_stTmp.rMasterPos           := _mcMotionFunctionPoint.MasterPos;
_stTmp.rSlavePos            := _mcMotionFunctionPoint.SlavePos;
_stTmp.rSlaveAcc            := _mcMotionFunctionPoint.SlaveAcc;
_stTmp.rSlaveJerk           := _mcMotionFunctionPoint.SlaveJerk;
_stTmp.rSlaveVelo           := _mcMotionFunctionPoint.SlaveVelo;

ReadMotionFunctionPointData := _stTmp;
END_GET
END_PROPERTY

METHOD ReadMotionFunctionValues : E_PROGRESS
VAR_INPUT
  Execute           : BOOL;
END_VAR
VAR_INST
  _eState           : E_PROGRESS;
  _rValue           : LREAL;
  _udiErr           : UDINT;
  _stMsg            : ST_Message;
END_VAR

IF NOT Execute THEN _eState   := E_PROGRESS.INIT; END_IF


CASE _eState
OF
  E_PROGRESS.INIT:
    IF Execute 
    THEN
      memset(ADR(_mcMotionFunction),0,SIZEOF(_mcMotionFunction));
      memset(ADR(_stMsg),0,SIZEOF(_stMsg));
      _udiErr                       := 0;
      _rValue                       := 0;
      _eState                       := E_PROGRESS.BUSY;

      _mcCamRef.pArray              := ADR(_mcMotionFunction);
      _mcCamRef.ArraySize           := SIZEOF(_mcMotionFunction);

      _mcCamRef.TableType           := Tc2_MC2_Camming.MC_TABLETYPE_MOTIONFUNCTION;
      _mcCamRef.NoOfColumns         := 1;

      _fbReadMotionFunctionValues(
              Execute               := FALSE, 
              CamTableID            := _stCamData.nCamTableId, 
              ValueSelectMask       := _stCamData.stReadValuesParameter.nValueSelectMask, 
              StartPosMaster        := _stCamData.stReadValuesParameter.rValueMasterStart, 
              EndPosMaster          := _stCamData.stReadValuesParameter.rValueMasterEnd, 
              Increment             := _stCamData.stReadValuesParameter.rIncrement, 
              CamTable              := _mcCamRef);
    END_IF
END_CASE
CASE _eState
OF
  E_PROGRESS.BUSY:
    _fbReadMotionFunctionValues(
              Execute               := TRUE, 
              CamTableID            := _stCamData.nCamTableId, 
              ValueSelectMask       := _stCamData.stReadValuesParameter.nValueSelectMask, 
              StartPosMaster        := _stCamData.stReadValuesParameter.rValueMasterStart, 
              EndPosMaster          := _stCamData.stReadValuesParameter.rValueMasterEnd, 
              Increment             := _stCamData.stReadValuesParameter.rIncrement, 
              CamTable              := _mcCamRef);

    IF (_fbReadMotionFunctionValues.Error)
    THEN
      _eState                       := E_PROGRESS.ERROR;
      _udiErr                       := _fbReadMotionFunctionValues.ErrorID;

      _stMsg.eType                  := E_MessageType.eMessageError;
      _stMsg.eDevice                := E_Device.Camming + TO_DINT(_AxisSlave.NcToPlc.AxisId);
      _stMsg.eSubdevice             := e_Subdevice.fbReadMotionFunctionValues;
      _stMsg.iErrorNumber           := _udiErr;

      _stMsg.sText                  := concat(' : ', TO_STRING(_eState));
      f_MessageSet(_stMsg);

      _fbReadMotionFunctionValues(
              Execute               := FALSE, 
              CamTableID            := _stCamData.nCamTableId, 
              ValueSelectMask       := _stCamData.stReadValuesParameter.nValueSelectMask, 
              StartPosMaster        := _stCamData.stReadValuesParameter.rValueMasterStart, 
              EndPosMaster          := _stCamData.stReadValuesParameter.rValueMasterEnd, 
              Increment             := _stCamData.stReadValuesParameter.rIncrement, 
              CamTable              := _mcCamRef);
    ELSE
      IF (_fbReadMotionFunctionValues.Done)
      THEN
        _eState                     := E_PROGRESS.DONE;
  
        _stMsg.eType                := E_MessageType.eMessageInfo;
        _stMsg.eDevice              := E_Device.Camming + TO_DINT(_AxisSlave.NcToPlc.AxisId);
        _stMsg.eSubdevice           := e_Subdevice.fbReadMotionFunctionValues;
        _stMsg.iErrorNumber         := 0;
  
        _stMsg.sText                := concat(' : ', TO_STRING(_eState));

        IF (_MessageLevel < E_MessageType.eMessageError)
        THEN
          f_MessageSet(_stMsg);
        END_IF
        _fbReadMotionFunctionValues(
              Execute               := FALSE, 
              CamTableID            := _stCamData.nCamTableId, 
              ValueSelectMask       := _stCamData.stReadValuesParameter.nValueSelectMask, 
              StartPosMaster        := _stCamData.stReadValuesParameter.rValueMasterStart, 
              EndPosMaster          := _stCamData.stReadValuesParameter.rValueMasterEnd, 
              Increment             := _stCamData.stReadValuesParameter.rIncrement, 
              CamTable              := _mcCamRef);
      END_IF
    END_IF
END_CASE

ReadMotionFunctionValues            := _eState;
END_METHOD

METHOD SetOnLineChangeMode : E_PROGRESS
VAR_INPUT
  Execute           : BOOL;
END_VAR
VAR_INST
  _eState           : E_PROGRESS;
  _rValue           : LREAL;
  _udiErr           : UDINT;
  _stMsg            : ST_Message;

  _nCopySize        : UINT;

END_VAR

IF NOT Execute THEN _eState   := E_PROGRESS.INIT; END_IF


CASE _eState
OF
  E_PROGRESS.INIT:
    IF Execute 
    THEN
      memset(ADR(_stMsg),0,SIZEOF(_stMsg));
      _udiErr                       := 0;
      _rValue                       := 0;
      _eState                       := E_PROGRESS.BUSY;

      _fbSetCamOnlineChangeMode(
              Execute               := FALSE, 
              ActivationMode        := _stCamData.nActivationMode, 
              ActivationPosition    := _stCamData.rActivationPosition, 
              MasterScalingMode     := _stCamData.stCamScalingData.nMasterScalingMode, 
              SlaveScalingMode      := _stCamData.stCamScalingData.nSlaveScalingMode, 
              CamTableID            := _stCamData.nCamTableId);
    END_IF
END_CASE
CASE _eState
OF
  E_PROGRESS.BUSY:
    _fbSetCamOnlineChangeMode(
              Execute               := TRUE, 
              ActivationMode        := _stCamData.nActivationMode, 
              ActivationPosition    := _stCamData.rActivationPosition, 
              MasterScalingMode     := _stCamData.stCamScalingData.nMasterScalingMode, 
              SlaveScalingMode      := _stCamData.stCamScalingData.nSlaveScalingMode, 
              CamTableID            := _stCamData.nCamTableId);

    IF (_fbSetCamOnlineChangeMode.Error)
    THEN
      _eState                       := E_PROGRESS.ERROR;
      _udiErr                       := _fbSetCamOnlineChangeMode.ErrorID;

      _stMsg.eType                  := E_MessageType.eMessageError;
      _stMsg.eDevice                := E_Device.Camming + TO_DINT(_AxisSlave.NcToPlc.AxisId);
      _stMsg.eSubdevice             := e_Subdevice.fbSetOnlineChangeMode;
      _stMsg.iErrorNumber           := _udiErr;

      _stMsg.sText                  := concat(' : ', TO_STRING(_eState));
      f_MessageSet(_stMsg);

      _fbSetCamOnlineChangeMode(
              Execute               := FALSE); 

    ELSIF (_fbSetCamOnlineChangeMode.Done)
    THEN
      _eState                       := E_PROGRESS.DONE;

      _stMsg.eType                  := E_MessageType.eMessageInfo;
      _stMsg.eDevice                := E_Device.Camming + TO_DINT(_AxisSlave.NcToPlc.AxisId);
      _stMsg.eSubdevice             := e_Subdevice.fbSetOnlineChangeMode;
      _stMsg.iErrorNumber           := 0;

      _stMsg.sText                  := concat(' : ', TO_STRING(_eState));

      IF (_MessageLevel < E_MessageType.eMessageError)
      THEN
        f_MessageSet(_stMsg);
      END_IF

      _fbSetCamOnlineChangeMode(
              Execute               := FALSE); 
    END_IF
END_CASE

SetOnLineChangeMode                 := _eState;
END_METHOD

METHOD Template : E_PROGRESS
VAR_INPUT
  Execute           : BOOL;
END_VAR
VAR_INST
  _eState           : E_PROGRESS;
  _rValue           : LREAL;
  _udiErr           : UDINT;
  _stMsg            : ST_Message;


END_VAR

IF NOT __ISVALIDREF(_AxisSlave)
THEN
  _eCheck                     := E_CHECK_STATE.CAM_SLAVE_AXIS_REF_INVALID;
  CamOut                      := E_PROGRESS.ERROR;
  RETURN;
END_IF

IF NOT Execute THEN _eState := E_PROGRESS.INIT; END_IF

CASE _eState
OF
  E_PROGRESS.INIT:
    IF Execute 
    THEN
      memset(ADR(_stMsg),0,SIZEOF(_stMsg));
      _udiErr                       := 0;
      _rValue                       := 0;
      _eState                       := E_PROGRESS.BUSY;
    END_IF
END_CASE
CASE _eState
OF
  E_PROGRESS.BUSY:
    _eState                         := E_PROGRESS.STARTUP;
END_CASE
CASE _eState
OF
  E_PROGRESS.STARTUP:
    _eState                         := E_PROGRESS.PREPARE;
END_CASE
CASE _eState
OF
  E_PROGRESS.PREPARE:
    _eState                         := E_PROGRESS.READY;
END_CASE
CASE _eState
OF
  E_PROGRESS.READY:
    _eState                         := E_PROGRESS.WAITING;
END_CASE
CASE _eState
OF
  E_PROGRESS.WAITING:
    _eState                         := E_PROGRESS.WORKING;
END_CASE
CASE _eState
OF
  E_PROGRESS.WORKING:
    _eState                         := E_PROGRESS.DONE;
END_CASE

Template_1 := _eState;
END_METHOD

METHOD WriteMotionFunction : E_PROGRESS
VAR_INPUT
  Execute           : BOOL;
END_VAR
VAR_INST
  _eResult,
  _eState           : E_PROGRESS;
  _rValue           : LREAL;
  _udiErr           : UDINT;
  _stMsg            : ST_Message;


END_VAR
IF NOT __ISVALIDREF(_AxisSlave)
THEN
  _eCheck                     := E_CHECK_STATE.CAM_SLAVE_AXIS_REF_INVALID;
  WriteMotionFunction         := E_PROGRESS.ERROR;
  RETURN;
END_IF

IF NOT Execute THEN _eState := E_PROGRESS.INIT; END_IF

CASE _eState
OF
  E_PROGRESS.INIT:
    IF Execute 
    THEN
      memset(ADR(_stMsg),0,SIZEOF(_stMsg));
      _udiErr                       := 0;
      _rValue                       := 0;
      _eState                       := E_PROGRESS.BUSY;
      _eResult                      := SetOnLineChangeMode(FALSE);
    END_IF
END_CASE
CASE _eState
OF
  E_PROGRESS.BUSY:
    _eResult                        := SetOnLineChangeMode(TRUE);
    IF (_eResult = E_PROGRESS.ERROR)
    THEN
      SetOnLineChangeMode(FALSE);
      _eState                       := E_PROGRESS.ERROR;
    ELSE
      IF (_eResult = E_PROGRESS.DONE)
      THEN
        SetOnLineChangeMode(FALSE);
        _eState                     := E_PROGRESS.STARTUP;
(*
        _mcMotionFunction           := _stMotionFunction.stMotionFunction;
*)
      END_IF
    END_IF
END_CASE
CASE _eState
OF
  E_PROGRESS.STARTUP:
    _eState                         := E_PROGRESS.WORKING;

    _mcCamRef.pArray                := ADR(_mcMotionFunction);
    _mcCamRef.ArraySize             := SIZEOF(_mcMotionFunction);

    _mcCamRef.TableType             := Tc2_MC2_Camming.MC_TABLETYPE_MOTIONFUNCTION;
    _mcCamRef.NoOfColumns           := 1;

    _fbWriteMotionFunction(
                    Execute         := FALSE, 
                    CamTableID      := _stCamData.nCamTableId, 
                    PointID         := _stCamData.nPointId, 
                    NumPoints       := _stCamData.nNumPoints, 
                    CamTable        := _mcCamRef);

END_CASE
CASE _eState
OF
  E_PROGRESS.WORKING:
    _fbWriteMotionFunction(
                    Execute         := TRUE, 
                    CamTableID      := _stCamData.nCamTableId, 
                    PointID         := _stCamData.nPointId, 
                    NumPoints       := _stCamData.nNumPoints, 
                    CamTable        := _mcCamRef);

    IF (_fbWriteMotionFunction.Error)
    THEN
      _eState                       := E_PROGRESS.ERROR;
      _udiErr                       := _fbWriteMotionFunction.ErrorID;

      _stMsg.eType                  := E_MessageType.eMessageError;
      _stMsg.eDevice                := E_Device.Camming + TO_DINT(_AxisSlave.NcToPlc.AxisId);
      _stMsg.eSubdevice             := e_Subdevice.fbWriteMotionFunction;
      _stMsg.iErrorNumber           := _udiErr;

      _stMsg.sText                  := concat(' : ', TO_STRING(_eState));
      f_MessageSet(_stMsg);

      _fbWriteMotionFunction(
                    Execute         := FALSE, 
                    CamTableID      := _stCamData.nCamTableId, 
                    PointID         := _stCamData.nPointId, 
                    NumPoints       := _stCamData.nNumPoints, 
                    CamTable        := _mcCamRef);
    ELSE
      IF (_fbWriteMotionFunction.Done)
      THEN
        _eState                     := E_PROGRESS.FINISHING;
        _fbWriteMotionFunction(
                    Execute         := FALSE, 
                    CamTableID      := _stCamData.nCamTableId, 
                    PointID         := _stCamData.nPointId, 
                    NumPoints       := _stCamData.nNumPoints, 
                    CamTable        := _mcCamRef);
      END_IF
    END_IF
END_CASE
CASE _eState
OF
  E_PROGRESS.FINISHING:
    _eState                         := E_PROGRESS.DONE;

    _stMsg.eType                    := E_MessageType.eMessageInfo;
    _stMsg.eDevice                  := E_Device.Camming + TO_DINT(_AxisSlave.NcToPlc.AxisId);
    _stMsg.eSubdevice               := e_Subdevice.fbWriteMotionFunction;
    _stMsg.iErrorNumber             := 0;

    _stMsg.sText                    := concat(' : ', TO_STRING(_eState));

    IF (_MessageLevel < E_MessageType.eMessageError)
    THEN
      f_MessageSet(_stMsg);
    END_IF
END_CASE

WriteMotionFunction                 := _eState;
END_METHOD

PROPERTY WriteMotionFunctionData : ST_MOTION_FUNCTION
SET
VAR
  _idx        : UINT;
  _stMf       : ST_MOTION_FUNCTION;
END_VAR

_stMf                                           := WriteMotionFunctionData;
memset(ADR(_mcMotionFunction), 0, SIZEOF(_mcMotionFunction));

FOR _idx := 1 TO MAX_MOTION_FUNCTION_POINTS
DO
  IF NOT (_idx > _stMf.nPoints)
  THEN
    _mcMotionFunction[_idx].FunctionType        := TO_INT(_stMf.stMotionFunction[_idx].nFunctionType);
    _mcMotionFunction[_idx].PointIndex          := _stMf.stMotionFunction[_idx].nPointIndex;
    _mcMotionFunction[_idx].RelIndexNextPoint   := _stMf.stMotionFunction[_idx].nRelIndexNextPoint;

    _mcMotionFunction[_idx].PointType           := to_int(_stMf.stMotionFunction[_idx].wPointType);

    _mcMotionFunction[_idx].MasterPos           := _stMf.stMotionFunction[_idx].rMasterPos;
    _mcMotionFunction[_idx].SlavePos            := _stMf.stMotionFunction[_idx].rSlavePos;

    _mcMotionFunction[_idx].SlaveVelo           := _stMf.stMotionFunction[_idx].rSlaveVelo;
    _mcMotionFunction[_idx].SlaveAcc            := _stMf.stMotionFunction[_idx].rSlaveAcc;
    _mcMotionFunction[_idx].SlaveJerk           := _stMf.stMotionFunction[_idx].rSlaveJerk;
  END_IF
END_FOR
END_SET
END_PROPERTY

METHOD WriteMotionFunctionPoint : E_PROGRESS
VAR_INPUT
  Execute           : BOOL;
END_VAR
VAR_INST
  _eResult,
  _eState           : E_PROGRESS;
  _rValue           : LREAL;
  _udiErr           : UDINT;
  _stMsg            : ST_Message;


END_VAR
IF NOT __ISVALIDREF(_AxisSlave)
THEN
  _eCheck                     := E_CHECK_STATE.CAM_SLAVE_AXIS_REF_INVALID;
  WriteMotionFunctionPoint    := E_PROGRESS.ERROR;
  RETURN;
END_IF

IF NOT Execute THEN _eState := E_PROGRESS.INIT; END_IF

CASE _eState
OF
  E_PROGRESS.INIT:
    IF Execute 
    THEN
      memset(ADR(_stMsg),0,SIZEOF(_stMsg));
      _udiErr                       := 0;
      _rValue                       := 0;
      _eState                       := E_PROGRESS.BUSY;
      _eResult                      := SetOnLineChangeMode(FALSE);

      IF (_stCamData.nPointIndex < 1) OR
         (_stCamData.nPointIndex > MAX_MOTION_FUNCTION_POINTS)
      THEN
        _eState                     := E_PROGRESS.ERROR;
        _udiErr                     := _stCamData.nPointIndex;
  
        _stMsg.eType                := E_MessageType.eMessageError;
        _stMsg.eDevice              := E_Device.Camming + TO_DINT(_AxisSlave.NcToPlc.AxisId);
        _stMsg.eSubdevice           := e_Subdevice.fbWriteMotionFunctionPoint;
        _stMsg.iErrorNumber         := _udiErr;
  
        _stMsg.sText                  := concat('POINT INDEX NOT IN RANGE: ', TO_STRING(_eState));
        f_MessageSet(_stMsg);

      END_IF
    END_IF
END_CASE
CASE _eState
OF
  E_PROGRESS.BUSY:
    _eResult                        := SetOnLineChangeMode(TRUE);
    IF (_eResult = E_PROGRESS.ERROR)
    THEN
      SetOnLineChangeMode(FALSE);
      _eState                       := E_PROGRESS.ERROR;
    ELSE
      IF (_eResult = E_PROGRESS.DONE)
      THEN
        SetOnLineChangeMode(FALSE);
        _eState                     := E_PROGRESS.STARTUP;
(*
        _mcMotionFunction           := _stMotionFunction.stMotionFunction;
*)
        _mcMotionFunctionPoint      := _mcMotionFunction[_stCamData.nPointIndex];
      END_IF
    END_IF
END_CASE
CASE _eState
OF
  E_PROGRESS.STARTUP:
    _eState                         := E_PROGRESS.WORKING;
    _fbWriteMotionFunctionPoint(
                      Execute       := FALSE, 
                      CamTableID    := _stCamData.nCamTableId, 
                      PointID       := _stCamData.nPointId,
                      Point         := _mcMotionFunctionPoint);
END_CASE
CASE _eState
OF
  E_PROGRESS.WORKING:
    _fbWriteMotionFunctionPoint(
                      Execute       := TRUE, 
                      CamTableID    := _stCamData.nCamTableId, 
                      PointID       := _stCamData.nPointId,
                      Point         := _mcMotionFunctionPoint);

    IF (_fbWriteMotionFunctionPoint.Error)
    THEN
      _eState                       := E_PROGRESS.ERROR;
      _udiErr                       := _fbWriteMotionFunctionPoint.ErrorID;

      _stMsg.eType                  := E_MessageType.eMessageError;
      _stMsg.eDevice                := E_Device.Camming + TO_DINT(_AxisSlave.NcToPlc.AxisId);
      _stMsg.eSubdevice             := e_Subdevice.fbWriteMotionFunctionPoint;
      _stMsg.iErrorNumber           := _udiErr;

      _stMsg.sText                  := concat(' : ', TO_STRING(_eState));
      f_MessageSet(_stMsg);

      _fbWriteMotionFunctionPoint(
                      Execute       := FALSE, 
                      CamTableID    := _stCamData.nCamTableId, 
                      PointID       := _stCamData.nPointId,
                      Point         := _mcMotionFunctionPoint);

    ELSE
      IF (_fbWriteMotionFunctionPoint.Done)
      THEN
        _eState                     := E_PROGRESS.FINISHING;
        _fbWriteMotionFunctionPoint(
                      Execute       := FALSE, 
                      CamTableID    := _stCamData.nCamTableId, 
                      PointID       := _stCamData.nPointId,
                      Point         := _mcMotionFunctionPoint);
      END_IF
    END_IF
END_CASE
CASE _eState
OF
  E_PROGRESS.FINISHING:
    _eState                         := E_PROGRESS.DONE;

    _stMsg.eType                    := E_MessageType.eMessageInfo;
    _stMsg.eDevice                  := E_Device.Camming + TO_DINT(_AxisSlave.NcToPlc.AxisId);
    _stMsg.eSubdevice               := e_Subdevice.fbWriteMotionFunctionPoint;
    _stMsg.iErrorNumber             := 0;

    _stMsg.sText                    := concat(' : ', TO_STRING(_eState));

    IF (_MessageLevel < E_MessageType.eMessageError)
    THEN
      f_MessageSet(_stMsg);
    END_IF
END_CASE

WriteMotionFunctionPoint            := _eState;
END_METHOD

PROPERTY WriteMotionFunctionPointData : ST_MOTION_FUNCTION_POINT
SET
VAR
  _idx        : UINT;
  _stMf       : ST_MOTION_FUNCTION_POINT;
END_VAR

_stMf                                       := WriteMotionFunctionPointData;
memset(ADR(_mcMotionFunctionPoint), 0, SIZEOF(_mcMotionFunctionPoint));

_mcMotionFunctionPoint.FunctionType         := TO_INT(_stMf.nFunctionType);
_mcMotionFunctionPoint.PointIndex           := _stMf.nPointIndex;
_mcMotionFunctionPoint.RelIndexNextPoint    := _stMf.nRelIndexNextPoint;

_mcMotionFunctionPoint.PointType            := TO_INT(_stMf.wPointType);

_mcMotionFunctionPoint.MasterPos            := _stMf.rMasterPos;
_mcMotionFunctionPoint.SlavePos             := _stMf.rSlavePos;

_mcMotionFunctionPoint.SlaveVelo            := _stMf.rSlaveVelo;
_mcMotionFunctionPoint.SlaveAcc             := _stMf.rSlaveAcc;
_mcMotionFunctionPoint.SlaveJerk            := _stMf.rSlaveJerk;
END_SET
END_PROPERTY

END_FUNCTION_BLOCK

// ---- NCI/FB_NciChannelCtrl.TcPOU
(*
-------------------------------------------------------------------------------
	NCI Channel Control

  2020/05/20  HAUD  0.1     kinematic and NCI separation
  2022/10/22  HAUD  0.2     PLC_OPEN_DRIVE adaption
  2023/12/29  HAUD  0.3     PLC_STATE_DRIVE adaption
-------------------------------------------------------------------------------
*)

// This SOFTWARE is provided as an Exemple by THE PROVIDER "as is" and "with all faults." THE PROVIDER makes no 
// representations or warranties of any kind concerning the safety, suitability, lack of viruses, inaccuracies, 
// typographical errors, or other harmful components of this SOFTWARE. There are inherent dangers in the use of 
// any software, and you are solely responsible for determining whether this SOFTWARE is compatible with your 
// equipment and other software installed on your equipment. You are also solely responsible for the protection 
// of your equipment and backup of your data, and THE PROVIDER will not be liable for any damages you may suffer 
// in connection with using, modifying, or distributing this SOFTWARE.

FUNCTION_BLOCK FB_NciChannelCtrl EXTENDS FB_NciChannel IMPLEMENTS I_Nci_Ctrl
VAR
  _nChnId               : UINT;

  _eCtrl,
  _eCtrlOld             : E_NCI_CTRL;

  _eState               : E_NCI_STATE;

  _eInit,
  _eResult,
  _eResultOld           : E_PROGRESS;

  // control and state struct from outside world
  _Ctrl                 : POINTER TO ST_CTRL_NCI;
  _State                : POINTER TO ST_STATE_NCI;

  // M function to fetch for scope/debugging
  _MFuncScope           : POINTER TO ST_NCI_M_FUNC;

  _fPathVelo            : LREAL;
  _nBlockNo             : UDINT;
  _sProgLine            : STRING(100); 
  _nMFunc               : INT;
  _nStateItp            : UINT;
END_VAR

METHOD Check : BOOL
VAR_INST
 
END_VAR

IF NOT SUPER^.Check() THEN RETURN; END_IF

IF NOT (_Ctrl <> 0)
THEN
  _eCheck                     := E_CHECK_STATE.NCI_CTRL_POINTER_INVALID;
  RETURN;
END_IF

IF NOT (_State <> 0)
THEN
  _eCheck                     := E_CHECK_STATE.NCI_STATE_POINTER_INVALID;
  RETURN;
END_IF

IF NOT (_MFuncScope <> 0)
THEN
  _eCheck                     := E_CHECK_STATE.NCI_M_FUNC_POINTER_INVALID;
  RETURN;
END_IF

_eCheck                       := E_CHECK_STATE.CHECK_DONE;
Check                         := TRUE;
END_METHOD

PROPERTY ChnCtrl : pointer to ST_CTRL_NCI
SET
_Ctrl := ChnCtrl;
END_SET
END_PROPERTY

PROPERTY ChnId : udint
GET
ChnId := _NciChannelRef^.NcToPlc.ChnId;
END_GET
END_PROPERTY

PROPERTY ChnState : pointer to ST_STATE_NCI
SET
_State := ChnState;
END_SET
END_PROPERTY

//
//  Cmd
//    - gets state for ctrl
//    - prepare your commands here
//    - init what you have to here
//
//-------------------------------------------------------------------------------------
METHOD PRIVATE Cmd  : E_NCI_STATE
VAR_INPUT
  eCmd      : E_NCI_CTRL;
END_VAR
VAR_INST
  _estate   : E_NCI_STATE;
  _stMsg    : ST_Message;
END_VAR

CASE eCmd
OF
  E_NCI_CTRL.INIT:
    // check axis configuration, clear group, reset Itp
    _eInit := _eResult      := Ctrl_Init(FALSE);
    _eState                 := E_NCI_STATE.INIT;
ELSE
  IF NOT (_eInit = E_PROGRESS.DONE)
  THEN
    _eResult                := E_PROGRESS.ERROR;
  
    _stMsg.eType            := E_MessageType.eMessageError;
    _stMsg.eDevice          := E_Device.NciChannelCtrl + TO_DINT(ChnId);
    _stMsg.eSubdevice       := e_Subdevice.NciControl;
    _stMsg.iErrorNumber     := -1;
  
    _stMsg.sText          := 'eInit:';
    _stMsg.sText          := concat(_stMsg.sText, TO_STRING(_eInit));
    _stMsg.sText          := concat(_stMsg.sText, ': ');
    _stMsg.sText          := concat(_stMsg.sText, TO_STRING(_eResult));

    f_MessageSet(_stMsg);

  ELSE
    CASE eCmd
    OF
      E_NCI_CTRL.IDLE:
        _eResult                := Ctrl_Idle(FALSE);
        _eState                 := E_NCI_STATE.IDLE;
    
      E_NCI_CTRL.FEED_TABLE:
        // nothing implemented yet
        _eResult                := E_PROGRESS.NOT_EXIST;
        _eState                 := E_NCI_STATE.FEED_TABLE;
    
      E_NCI_CTRL.RESET:
        _eResult                := Ctrl_Reset(FALSE);
        _eState                 := E_NCI_STATE.RESET;
    
      E_NCI_CTRL.LOAD_PROG:
        _eResult                := Ctrl_LoadProg(FALSE);
        _eState                 := E_NCI_STATE.LOAD_PROG;
    
      E_NCI_CTRL.BUILD_GROUP:
        _eResult                := Ctrl_BuildGroup(FALSE);
        _eState                 := E_NCI_STATE.BUILD_GROUP;
    
      E_NCI_CTRL.CLEAR_GROUP:
        _eResult                := Ctrl_ClearGroup(FALSE);
        _eState                 := E_NCI_STATE.CLEAR_GROUP;
    
      E_NCI_CTRL.START:
        _eResult                := Ctrl_Start(FALSE);
        _eState                 := E_NCI_STATE.START;
    
      E_NCI_CTRL.STOP:
        _eResult                := Ctrl_Stop(FALSE);
        _eState                 := E_NCI_STATE.STOP;
    
      E_NCI_CTRL.STO_STOP:
        _eResult                := Ctrl_Stop_STO(FALSE);
        _eState                 := E_NCI_STATE.STO_STOP;
    
      E_NCI_CTRL.RESTART_STEP_ON:
        _eResult                := Ctrl_Restart(FALSE);
        _eState                 := E_NCI_STATE.RESTART_STEP_ON;
    
      E_NCI_CTRL.M_FUNC_QUIT:
        _eResult                := Ctrl_ConfirmHsk(FALSE);
        _eState                 := E_NCI_STATE.M_FUNC_QUIT;
    
      E_NCI_CTRL.READ_R_PARA:
        _eResult                := Ctrl_R_Parameter_Rd(FALSE);
        _eState                 := E_NCI_STATE.READ_R_PARA;
    
      E_NCI_CTRL.WRITE_R_PARA:
        _eResult                := Ctrl_R_Parameter_Wrt(FALSE);
        _eState                 := E_NCI_STATE.WRITE_R_PARA;
    ELSE
      _eState                 := E_NCI_STATE.NULL;
  
      IF (eCmd = E_NCI_CTRL.NULL)
      THEN
        _eResult              := E_PROGRESS.DONE;
      ELSE
        _eResult              := E_PROGRESS.INVALID;
  
        _stMsg.eType          := E_MessageType.eMessageError;
        _stMsg.eDevice        := E_Device.NciChannelCtrl + TO_DINT(ChnId);
        _stMsg.eSubdevice     := e_Subdevice.NciControl;
        _stMsg.iErrorNumber   := 0;
  
        _stMsg.sText          := 'E_NCI_CTRL.';
        _stMsg.sText          := concat(_stMsg.sText, TO_STRING(eCmd));
        _stMsg.sText          := concat(_stMsg.sText, ': ');
        _stMsg.sText          := concat(_stMsg.sText, TO_STRING(_eResult));
  
        f_MessageSet(_stMsg);
      END_IF
    END_CASE
  END_IF
END_CASE


Cmd                         := _eState;
END_METHOD

METHOD PRIVATE Ctrl_BuildGroup : E_PROGRESS
VAR_INPUT
  Execute           : BOOL;
END_VAR
VAR_INST
  _eJobResult,
  _eState           : E_PROGRESS;
END_VAR
IF NOT Check() THEN Ctrl_BuildGroup := E_PROGRESS.ERROR; RETURN; END_IF
IF NOT Execute THEN _eState := E_PROGRESS.INIT; END_IF

CASE _eState
OF
  E_PROGRESS.INIT:
    IF Execute 
    THEN
      _eJobResult                   := BuilDGroup(FALSE);
      _eState                       := E_PROGRESS.BUSY;
    END_IF
END_CASE
CASE _eState
OF
  E_PROGRESS.BUSY:
    _eJobResult                     := BuilDGroup(TRUE);

    IF (_eJobResult = E_PROGRESS.ERROR)
    THEN
      BuilDGroup(FALSE);
      _eState                       := E_PROGRESS.ERROR;

    ELSIF (_eJobResult = E_PROGRESS.DONE)
    THEN
      BuilDGroup(FALSE);
      _eState                       := E_PROGRESS.STARTUP;
    END_IF
END_CASE
CASE _eState
OF
  E_PROGRESS.STARTUP:
    _eState                         := E_PROGRESS.PREPARE;
END_CASE
CASE _eState
OF
  E_PROGRESS.PREPARE:
    _eState                         := E_PROGRESS.READY;
END_CASE
CASE _eState
OF
  E_PROGRESS.READY:
    _eState                         := E_PROGRESS.WAITING;
END_CASE
CASE _eState
OF
  E_PROGRESS.WAITING:
    _eState                         := E_PROGRESS.WORKING;
END_CASE
CASE _eState
OF
  E_PROGRESS.WORKING:
    _eState                         := E_PROGRESS.DONE;
END_CASE

Ctrl_BuildGroup                      := _eState;
END_METHOD

METHOD PRIVATE Ctrl_ClearGroup : E_PROGRESS
VAR_INPUT
  Execute           : BOOL;
END_VAR
VAR_INST
  _eJobResult,
  _eState           : E_PROGRESS;
END_VAR
IF NOT Check() THEN Ctrl_ClearGroup := E_PROGRESS.ERROR; RETURN; END_IF
IF NOT Execute THEN _eState := E_PROGRESS.INIT; END_IF

CASE _eState
OF
  E_PROGRESS.INIT:
    IF Execute 
    THEN
      _eJobResult                           := ClearGroup(FALSE);
      _eState                               := E_PROGRESS.BUSY;
    END_IF

  E_PROGRESS.BUSY:
    _eJobResult                             := ClearGroup(TRUE);
    IF (_eJobResult = E_PROGRESS.ERROR)
    THEN
      ClearGroup(FALSE);
      _eState                               := E_PROGRESS.ERROR;

    ELSIF (_eJobResult = E_PROGRESS.DONE)
    THEN
      ClearGroup(FALSE);
      _eJobResult                           := ItpReset(FALSE);
      _eState                               := E_PROGRESS.STARTUP;
    END_IF

  E_PROGRESS.STARTUP:
    _eJobResult                             := ItpReset(TRUE);
    IF (_eJobResult = E_PROGRESS.ERROR)
    THEN
      ItpReset(FALSE);
      _eState                               := E_PROGRESS.ERROR;

    ELSIF (_eJobResult = E_PROGRESS.DONE)
    THEN
      ItpReset(FALSE);
      _eState                               := E_PROGRESS.PREPARE;
    END_IF

  E_PROGRESS.PREPARE:
    IF (_NciChannelRef^.NcToPlc.HskMFuncReq = 0)
    THEN
      _eState                               := E_PROGRESS.DONE;
    ELSE
      _NciChannelRef^.PlcToNc.MFuncGranted  := 0;
      _eState                               := E_PROGRESS.READY;
    END_IF

  E_PROGRESS.READY:
      _NciChannelRef^.PlcToNc.MFuncGranted  := 1;
      _eState                               := E_PROGRESS.PREPARE;

  E_PROGRESS.DONE:
    _NciChannelRef^.PlcToNc.MFuncGranted    := 0;
END_CASE


Ctrl_ClearGroup                             := _eState;
END_METHOD

METHOD PRIVATE Ctrl_ConfirmHsk : E_PROGRESS
VAR_INPUT
  Execute           : BOOL;
END_VAR
VAR_INST
  _eJobResult,
  _eState           : E_PROGRESS;
END_VAR
IF NOT Check() THEN Ctrl_ConfirmHsk := E_PROGRESS.ERROR; RETURN; END_IF
IF NOT Execute THEN _eState := E_PROGRESS.INIT; END_IF

CASE _eState
OF
  E_PROGRESS.INIT:
    IF Execute 
    THEN
      _eJobResult                         := ConfirmHSK(FALSE);
      _eState                             := E_PROGRESS.BUSY;
    END_IF
END_CASE
CASE _eState
OF

  E_PROGRESS.BUSY:
    _eJobResult                           := ConfirmHSK(TRUE);

    IF (_eJobResult = E_PROGRESS.ERROR)
    THEN
      ConfirmHSK(FALSE);
      _eState                             := E_PROGRESS.ERROR;

    ELSIF (_eJobResult = E_PROGRESS.DONE)
    THEN
      ConfirmHSK(FALSE);
      _eState                             := E_PROGRESS.PREPARE;
    END_IF
END_CASE
CASE _eState
OF
  E_PROGRESS.PREPARE:
    _eState                               := E_PROGRESS.DONE;
END_CASE

Ctrl_ConfirmHsk                            := _eState;
END_METHOD

METHOD PRIVATE Ctrl_Idle : E_PROGRESS
VAR_INPUT
  Execute           : BOOL;
END_VAR
VAR_INST
  _eJobResult,
  _eState           : E_PROGRESS;

  _nErr             : DWORD;
  _NciAxisIds       : ARRAY[1..8] OF DWORD;

  _stMsg            : ST_Message;
END_VAR
IF NOT Check() THEN Ctrl_Idle := E_PROGRESS.ERROR; RETURN; END_IF
IF NOT Execute THEN _eState := E_PROGRESS.INIT; END_IF

CASE _eState
OF
  E_PROGRESS.INIT:
    IF Execute 
    THEN
      _eJobResult                         := ItpReset(FALSE);
      _eState                             := E_PROGRESS.BUSY;
    END_IF
END_CASE
CASE _eState
OF
  E_PROGRESS.BUSY:
    IF (_NciChannelRef^.NcToPlc.ItpState <> Tc2_NCI.NCI_INTERPRETER_IDLE)
    THEN
      _eState                             := E_PROGRESS.STARTUP;
    ELSE
      IF (_NciChannelRef^.PlcToNc.ChnAxesOvr > 0) AND NOT
         (_NciChannelRef^.NcToPlc.ChnState.8)
      THEN
        _eState                           := E_PROGRESS.PREPARE;
      END_IF
    END_IF
END_CASE
CASE _eState
OF
  E_PROGRESS.STARTUP:
    _eJobResult                           := ItpReset(TRUE);
    IF (_eJobResult = E_PROGRESS.ERROR)
    THEN
      ItpReset(FALSE);
      _eState                             := E_PROGRESS.ERROR;

    ELSIF (_eJobResult = E_PROGRESS.DONE)
    THEN
      ItpReset(FALSE);
      _eState                             := E_PROGRESS.PREPARE;
    END_IF

  E_PROGRESS.PREPARE:
    _NciChannelRef^.PlcToNc.MFuncGranted  := 0;
    _eState                               := E_PROGRESS.READY;

END_CASE
CASE _eState
OF
  E_PROGRESS.READY:
    _nErr                                 := ItpGetGroupAxisIds(_NciAxisIds, _NciChannelRef^.NcToPlc);

    IF (_NciChannelRef^.NcToPlc.HskMFuncReq = 0)
    THEN
      IF (_nErr <> 0)
      THEN
        _eState                           := E_PROGRESS.ERROR;
        _stMsg.eType                      := E_MessageType.eMessageError;
        _stMsg.eDevice                    := ChannelDevice;
        _stMsg.eSubdevice                 := e_Subdevice.NciIdle;
        _stMsg.iErrorNumber               := _nErr;
        _stMsg.sText                      := concat('ItpGetGroupAxisIds Error: ', TO_STRING(_nErr));

        f_MessageSet(_stMsg);
      ELSE
        _eState                           := E_PROGRESS.DONE;
      END_IF
    ELSE
      _eState                             := E_PROGRESS.STARTUP;
    END_IF
END_CASE

Ctrl_Idle                                := _eState;
END_METHOD

METHOD Ctrl_Init : E_PROGRESS
VAR_INPUT
  Execute           : BOOL;
END_VAR
VAR_INST
  _eJobResult,
  _eState           : E_PROGRESS;
  _rValue           : LREAL;
  _udiErr           : UDINT;

  _nErr             : DWORD;
  _NciAxisIds       : ARRAY[1..8] OF DWORD;

  _stMsg            : ST_Message;
END_VAR
IF NOT Check() THEN _eState := E_PROGRESS.ERROR; END_IF
IF NOT Execute THEN _eState := E_PROGRESS.INIT; END_IF

CASE _eState
OF
  E_PROGRESS.INIT:
    IF Execute 
    THEN
      memset(ADR(_stMsg),0,SIZEOF(_stMsg));
      _udiErr                       := 0;
      _rValue                       := 0;
      _eState                       := E_PROGRESS.BUSY;
    END_IF
END_CASE
CASE _eState
OF
  E_PROGRESS.BUSY:
    IF NOT (_stCfgAxes^.nXAxisId > 0) OR
       NOT (_stCfgAxes^.nYAxisId > 0) OR
       NOT (_stCfgAxes^.nZAxisId > 0)
    THEN
      _eState                       := E_PROGRESS.WAITING;

      _stMsg.eType                  := E_MessageType.eMessageWarn;
      _stMsg.eDevice                := ChannelDevice;
      _stMsg.eSubdevice             := e_Subdevice.NciStartUp;
      _stMsg.iErrorNumber           := _eState;
      _stMsg.sText                  := concat('Init NCI channel AxisConfig: ', TO_STRING(_eState));

      f_MessageSet(_stMsg);
    ELSE
      _eJobResult                   := ItpReset(FALSE);
      _eState                       := E_PROGRESS.STARTUP;
    END_IF
END_CASE
CASE _eState
OF
  E_PROGRESS.STARTUP:
    _eJobResult                     := ItpReset(TRUE);
    IF (_eJobResult = E_PROGRESS.ERROR)
    THEN
      _eState                       := E_PROGRESS.ERROR;
    ELSIF (_eJobResult = E_PROGRESS.DONE)
    THEN
      _eJobResult                   := ItpReset  (FALSE);
      _eJobResult                   := ClearGroup(FALSE);
      _eState                       := E_PROGRESS.PREPARE;
    END_IF
END_CASE
CASE _eState
OF
  E_PROGRESS.PREPARE:
    _eJobResult                     := ClearGroup(TRUE);
    IF (_eJobResult = E_PROGRESS.ERROR)
    THEN
      _eState                       := E_PROGRESS.ERROR;
    ELSIF (_eJobResult = E_PROGRESS.DONE)
    THEN
      _eJobResult                   := ClearGroup(FALSE);
      _eState                       := E_PROGRESS.READY;
    END_IF

END_CASE
CASE _eState
OF
  E_PROGRESS.READY:
    _eState                         := E_PROGRESS.WORKING;
END_CASE
CASE _eState
OF
  E_PROGRESS.WAITING:
    IF (_stCfgAxes^.nXAxisId > 0) AND
       (_stCfgAxes^.nYAxisId > 0) AND
       (_stCfgAxes^.nZAxisId > 0)
    THEN
      _eState                       := E_PROGRESS.STARTUP;

      _stMsg.eType                  := E_MessageType.eMessageInfo;
      _stMsg.eDevice                := ChannelDevice;
      _stMsg.eSubdevice             := e_Subdevice.NciStartUp;
      _stMsg.iErrorNumber           := _eState;
      _stMsg.sText                  := concat('Init NCI channel AxisConfig: ', TO_STRING(_eState));

      IF (_MessageLevel < E_MessageType.eMessageError)
      THEN
        f_MessageSet(_stMsg);
      END_IF
    END_IF
END_CASE
CASE _eState
OF
  E_PROGRESS.WORKING:
    _eState                         := E_PROGRESS.DONE;
END_CASE

Ctrl_Init                           := _eState;
END_METHOD

METHOD PRIVATE Ctrl_LoadProg : E_PROGRESS
VAR_INPUT
  Execute           : BOOL;
END_VAR
VAR_INST
  _eJobResult,
  _eState           : E_PROGRESS;
END_VAR
IF NOT Check() THEN Ctrl_LoadProg := E_PROGRESS.ERROR; RETURN; END_IF
IF NOT Execute THEN _eState := E_PROGRESS.INIT; END_IF

CASE _eState
OF
  E_PROGRESS.INIT:
    IF Execute 
    THEN
      _eJobResult                         := LoadProg(FALSE);
      _eState                             := E_PROGRESS.BUSY;
    END_IF

  E_PROGRESS.BUSY:
    _NciChannelRef^.PlcToNc.MFuncGranted  := 0;
    _eJobResult                           := LoadProg(TRUE);

    IF (_eJobResult = E_PROGRESS.ERROR)
    THEN
      LoadProg(FALSE);
      _eState                             := E_PROGRESS.ERROR;

    ELSIF (_eJobResult = E_PROGRESS.DONE)
    THEN
      LoadProg(FALSE);
      _eState                             := E_PROGRESS.DONE;
    END_IF
END_CASE

Ctrl_LoadProg                      := _eState;
END_METHOD

METHOD PRIVATE Ctrl_R_Parameter_Rd : E_PROGRESS
VAR_INPUT
  Execute           : BOOL;
END_VAR
VAR_INST
  _eJobResult,
  _eState           : E_PROGRESS;
END_VAR
IF NOT Check() THEN Ctrl_R_Parameter_Rd := E_PROGRESS.ERROR; RETURN; END_IF
IF NOT Execute THEN _eState := E_PROGRESS.INIT; END_IF

CASE _eState
OF
  E_PROGRESS.INIT:
    IF Execute 
    THEN
      _eJobResult                         := ReadRParams(FALSE);
      _eState                             := E_PROGRESS.BUSY;
    END_IF

  E_PROGRESS.BUSY:
    _NciChannelRef^.PlcToNc.MFuncGranted  := 0;
    _eJobResult                           := ReadRParams(TRUE);

    IF (_eJobResult = E_PROGRESS.ERROR)
    THEN
      ReadRParams(FALSE);
      _eState                             := E_PROGRESS.ERROR;

    ELSIF (_eJobResult = E_PROGRESS.DONE)
    THEN
      ReadRParams(FALSE);
      _eState                             := E_PROGRESS.STARTUP;
    END_IF
END_CASE
CASE _eState
OF
  E_PROGRESS.STARTUP:
    _NciChannelRef^.PlcToNc.MFuncGranted  := 1;
    _eState                               := E_PROGRESS.PREPARE;

  E_PROGRESS.PREPARE:
    _NciChannelRef^.PlcToNc.MFuncGranted  := 0;
    _eState                               := E_PROGRESS.DONE;
END_CASE

Ctrl_R_Parameter_Rd                       := _eState;
END_METHOD

METHOD PRIVATE Ctrl_R_Parameter_Wrt : E_PROGRESS
VAR_INPUT
  Execute           : BOOL;
END_VAR
VAR_INST
  _eJobResult,
  _eState           : E_PROGRESS;
END_VAR
IF NOT Check() THEN Ctrl_R_Parameter_Wrt := E_PROGRESS.ERROR; RETURN; END_IF
IF NOT Execute THEN _eState := E_PROGRESS.INIT; END_IF

CASE _eState
OF
  E_PROGRESS.INIT:
    IF Execute 
    THEN
      _eJobResult                         := WriteRParams(FALSE);
      _eState                             := E_PROGRESS.BUSY;
    END_IF

  E_PROGRESS.BUSY:
    _NciChannelRef^.PlcToNc.MFuncGranted  := 0;
    _eJobResult                           := WriteRParams(TRUE);

    IF (_eJobResult = E_PROGRESS.ERROR)
    THEN
      WriteRParams(FALSE);
      _eState                             := E_PROGRESS.ERROR;

    ELSIF (_eJobResult = E_PROGRESS.DONE)
    THEN
      WriteRParams(FALSE);
      _eState                             := E_PROGRESS.STARTUP;
    END_IF
END_CASE
CASE _eState
OF
  E_PROGRESS.STARTUP:
    _NciChannelRef^.PlcToNc.MFuncGranted  := 1;
    _eState                               := E_PROGRESS.PREPARE;

  E_PROGRESS.PREPARE:
    _NciChannelRef^.PlcToNc.MFuncGranted  := 0;
    _eState                               := E_PROGRESS.DONE;
END_CASE

Ctrl_R_Parameter_Wrt                      := _eState;
END_METHOD

METHOD PRIVATE Ctrl_Reset : E_PROGRESS
VAR_INPUT
  Execute           : BOOL;
END_VAR
VAR_INST
  _eJobResult,
  _eState           : E_PROGRESS;
END_VAR
IF NOT Check() THEN Ctrl_Reset := E_PROGRESS.ERROR; RETURN; END_IF
IF NOT Execute THEN _eState := E_PROGRESS.INIT; END_IF

CASE _eState
OF
  E_PROGRESS.INIT:
    IF Execute 
    THEN
      _eJobResult                         := ItpReset(FALSE);
      _eState                             := E_PROGRESS.BUSY;
    END_IF
END_CASE
CASE _eState
OF
  E_PROGRESS.BUSY:
    _NciChannelRef^.PlcToNc.MFuncGranted  := 0;
    _eJobResult                           := ItpReset(TRUE);

    IF (_eJobResult = E_PROGRESS.ERROR)
    THEN
      ItpReset(FALSE);
      _eState                             := E_PROGRESS.ERROR;

    ELSIF (_eJobResult = E_PROGRESS.DONE)
    THEN
      ItpReset(FALSE);
      _eState                             := E_PROGRESS.STARTUP;
    END_IF

  E_PROGRESS.STARTUP:
    _NciChannelRef^.PlcToNc.MFuncGranted  := 1;
    _eState                               := E_PROGRESS.PREPARE;

  E_PROGRESS.PREPARE:
    _NciChannelRef^.PlcToNc.MFuncGranted  := 0;
    _eState                               := E_PROGRESS.READY;

END_CASE
CASE _eState
OF
  E_PROGRESS.READY:
    IF (_NciChannelRef^.NcToPlc.HskMFuncReq = 0)
    THEN
      _eState                             := E_PROGRESS.DONE;
    ELSE
      _eState                             := E_PROGRESS.STARTUP;
    END_IF
END_CASE

Ctrl_Reset                                := _eState;
END_METHOD

METHOD PRIVATE Ctrl_Restart : E_PROGRESS
VAR_INPUT
  Execute           : BOOL;
END_VAR
VAR_INST
  _eJobResult,
  _eState           : E_PROGRESS;
END_VAR
IF NOT Check() THEN Ctrl_Restart := E_PROGRESS.ERROR; RETURN; END_IF
IF NOT Execute THEN _eState := E_PROGRESS.INIT; END_IF

CASE _eState
OF
  E_PROGRESS.INIT:
    IF Execute 
    THEN
      _eJobResult                         := StepOnAfterEStop(FALSE);
      _eState                             := E_PROGRESS.BUSY;
    END_IF
END_CASE
CASE _eState
OF
  E_PROGRESS.BUSY:
    _NciChannelRef^.PlcToNc.MFuncGranted  := 0;
    _eJobResult                           := StepOnAfterEStop(TRUE);

    IF (_eJobResult = E_PROGRESS.ERROR)
    THEN
      StepOnAfterEStop(FALSE);
      _eState                             := E_PROGRESS.ERROR;

    ELSIF (_eJobResult = E_PROGRESS.DONE)
    THEN
      StepOnAfterEStop(FALSE);
      _eState                             := E_PROGRESS.DONE;
    END_IF
END_CASE


Ctrl_Restart                              := _eState;
END_METHOD

METHOD PRIVATE Ctrl_Start : E_PROGRESS
VAR_INPUT
  Execute           : BOOL;
END_VAR
VAR_INST
  _eJobResult,
  _eState           : E_PROGRESS;
END_VAR
IF NOT Check() THEN Ctrl_Start := E_PROGRESS.ERROR; RETURN; END_IF
IF NOT Execute THEN _eState := E_PROGRESS.INIT; END_IF

CASE _eState
OF
  E_PROGRESS.INIT:
    IF Execute 
    THEN
      _eJobResult                         := StartStop(FALSE, TRUE, FALSE);
      _eState                             := E_PROGRESS.BUSY;
    END_IF
END_CASE
CASE _eState
OF
  E_PROGRESS.BUSY:
    _NciChannelRef^.PlcToNc.MFuncGranted  := 0;
    _eJobResult                           := StartStop(TRUE, TRUE, FALSE);

    IF (_eJobResult = E_PROGRESS.ERROR)
    THEN
      StartStop(FALSE, TRUE, FALSE);
      _eState                             := E_PROGRESS.ERROR;

    ELSIF (_eJobResult = E_PROGRESS.DONE)
    THEN
      StartStop(FALSE, TRUE, FALSE);
      _eState                             := E_PROGRESS.DONE;
    END_IF
END_CASE

Ctrl_Start                                := _eState;
END_METHOD

METHOD PRIVATE Ctrl_Stop : E_PROGRESS
VAR_INPUT
  Execute           : BOOL;
END_VAR
VAR_INST
  _eJobResult,
  _eState           : E_PROGRESS;
END_VAR
IF NOT Check() THEN Ctrl_Stop := E_PROGRESS.ERROR; RETURN; END_IF
IF NOT Execute THEN _eState := E_PROGRESS.INIT; END_IF

CASE _eState
OF
  E_PROGRESS.INIT:
    IF Execute 
    THEN
      _eJobResult                         := StartStop(FALSE, FALSE, TRUE);
      _eState                             := E_PROGRESS.BUSY;
    END_IF
END_CASE
CASE _eState
OF
  E_PROGRESS.BUSY:
    _NciChannelRef^.PlcToNc.MFuncGranted  := 0;
    _eJobResult                           := StartStop(TRUE, FALSE, TRUE);

    IF (_eJobResult = E_PROGRESS.ERROR)
    THEN
      StartStop(FALSE, FALSE, TRUE);
      _eState                             := E_PROGRESS.ERROR;

    ELSIF (_eJobResult = E_PROGRESS.DONE)
    THEN
      StartStop(FALSE, FALSE, TRUE);
      _eState                             := E_PROGRESS.DONE;
    END_IF
END_CASE

Ctrl_Stop                                := _eState;
END_METHOD

METHOD PRIVATE Ctrl_Stop_STO : E_PROGRESS
VAR_INPUT
  Execute           : BOOL;
END_VAR
VAR_INST
  _eJobResult,
  _eState           : E_PROGRESS;
END_VAR
IF NOT Check() THEN Ctrl_Stop_STO := E_PROGRESS.ERROR; RETURN; END_IF
IF NOT Execute THEN _eState := E_PROGRESS.INIT; END_IF

CASE _eState
OF
  E_PROGRESS.INIT:
    IF Execute 
    THEN
      _eJobResult                         := EStop(FALSE);
      _eState                             := E_PROGRESS.BUSY;
    END_IF
END_CASE
CASE _eState
OF
  E_PROGRESS.BUSY:
    _NciChannelRef^.PlcToNc.MFuncGranted  := 0;
    _eJobResult                           := EStop(TRUE);

    IF (_eJobResult = E_PROGRESS.ERROR)
    THEN
      EStop(FALSE);
      _eState                             := E_PROGRESS.ERROR;

    ELSIF (_eJobResult = E_PROGRESS.DONE)
    THEN
      EStop(FALSE);
      _eState                             := E_PROGRESS.DONE;
    END_IF
END_CASE

Ctrl_Stop_STO                                := _eState;
END_METHOD

METHOD Cycle  : e_progress
VAR_INST
  _eCycle     : E_PROGRESS;
END_VAR

IF NOT Check() THEN Cycle := _eCycle := _eResult := E_PROGRESS.ERROR; RETURN; END_IF

ChannelDevice := e_Device.NciChannel + TO_UINT(ChnId);
//-----------------------------------------------------------------------------
//-----------------------------------------------------------------------------
// cyclic data for M func from NCI interface
//-----------------------------------------------------------------------------
_MFuncScope^.FastMFuncMask    := _NciChannelRef^.NcToPlc.FastMFuncMask;
_MFuncScope^.HskMFuncNo       := _NciChannelRef^.NcToPlc.HskMFuncNo;
_MFuncScope^.HskMFuncReq      := _NciChannelRef^.NcToPlc.HskMFuncReq;
_MFuncScope^.HFuncValue       := _NciChannelRef^.NcToPlc.HFuncValue;
_MFuncScope^.MFuncGranted     := _NciChannelRef^.PlcToNc.MFuncGranted;
//-----------------------------------------------------------------------------
//-----------------------------------------------------------------------------
// M-Func to catch
//-----------------------------------------------------------------------------
IF HSK 
THEN
  _nMFunc := MFunc;
END_IF
//-----------------------------------------------------------------------------
//-----------------------------------------------------------------------------
_eCtrl                         := _Ctrl^.eCmd;
//-----------------------------------------------------------------------------
//-----------------------------------------------------------------------------
// cmd change
//-----------------------------------------------------------------------------
IF (_eCtrl <> _eCtrlOld)
THEN
  LogControl();
  _eState                     := Cmd(_eCtrl);
  _eCtrlOld                   := _eCtrl;
END_IF
//-----------------------------------------------------------------------------
//-----------------------------------------------------------------------------
CASE _eResult
OF
  E_PROGRESS.INVALID:
    _State^.eState            := TO_UINT(E_PROGRESS.ERROR);

  E_PROGRESS.ERROR:
    _State^.eState            := _eState + E_PROGRESS.ERROR;

  E_PROGRESS.DONE:
    _State^.eState            := _eState + E_PROGRESS.DONE;

ELSE
    _State^.eState            := _eState + _eResult;
  CASE _eState
  OF
  E_NCI_STATE.INIT:
    _eResult      := _eInit   := Ctrl_Init(TRUE);

  E_NCI_STATE.IDLE:
    _eResult                  := Ctrl_Idle(TRUE);

  E_NCI_STATE.RESET:
    _eResult                  := Ctrl_Reset(TRUE);

  E_NCI_STATE.LOAD_PROG:
    _eResult                  := Ctrl_LoadProg(TRUE);

  E_NCI_STATE.BUILD_GROUP:
    _eResult                  := Ctrl_BuildGroup(TRUE);

  E_NCI_STATE.CLEAR_GROUP:
    _eResult                  := Ctrl_ClearGroup(TRUE);

  E_NCI_STATE.START:
    _eResult                  := Ctrl_Start(TRUE);

  E_NCI_STATE.STOP:
    _eResult                  := Ctrl_Stop(TRUE);

  E_NCI_STATE.STO_STOP:
    _eResult                  := Ctrl_Stop_STO(TRUE);

  E_NCI_STATE.RESTART_STEP_ON:
    _eResult                  := Ctrl_Restart(TRUE);

  E_NCI_STATE.M_FUNC_QUIT:
    _eResult                  := Ctrl_ConfirmHsk(TRUE);

  E_NCI_STATE.READ_R_PARA:
    _eResult                  := Ctrl_R_Parameter_Rd(TRUE);

  E_NCI_STATE.WRITE_R_PARA:
    _eResult                  := Ctrl_R_Parameter_Wrt(TRUE);
  END_CASE
END_CASE
//-----------------------------------------------------------------------------
//-----------------------------------------------------------------------------
//  OnChange of execution state result
//    - log result
//-----------------------------------------------------------------------------
IF (_eResult <> _eResultOld)
THEN
  LogResult();
  _eResultOld                 := _eResult;
END_IF
//-----------------------------------------------------------------------------
//-----------------------------------------------------------------------------
//  cyclic data from ChannelRef
//-----------------------------------------------------------------------------
_State^.rAxisOverride         := _NciChannelRef^.PlcToNc.ChnAxesOvr;
_State^.bMFuncReq             := TO_BOOL(_NciChannelRef^.NcToPlc.HskMFuncReq);
_State^.nMFunc                := _NciChannelRef^.NcToPlc.HskMFuncNo;
_State^.nItpState             := GetItpState();
//-----------------------------------------------------------------------------
//-----------------------------------------------------------------------------
Cycle := _eCycle              := E_PROGRESS.WORKING;
END_METHOD

PROPERTY ItfChannel : I_NciChannel
GET
ItfChannel := SUPER^;
END_GET
END_PROPERTY

METHOD LogControl
VAR_INST
  _sResult,
  _sCtrl            : STRING(30);

  _stMsg            : ST_Message;
END_VAR
  _stMsg.eType               := E_MessageType.eMessageInfo;
  _stMsg.eDevice             := E_Device.NciChannelCtrl + TO_UINT(ChnId);
  _stMsg.eSubdevice          := e_Subdevice.NciControl;
  _stMsg.iErrorNumber        := 0;

  _sCtrl                     := concat('E_NCI_CTRL', '.');
  _sCtrl                     := concat(_sCtrl, TO_STRING(_eCtrl));

  _stMsg.sText               := concat('new command: ', _sCtrl);

  IF (_MessageLevel < E_MessageType.eMessageError)
  THEN
    f_MessageSet(_stMsg);
  ELSE
    IF (_stMsg.eType = E_MessageType.eMessageError)
    THEN
      f_MessageSet(_stMsg);
    END_IF
  END_IF
END_METHOD

METHOD PRIVATE LogResult
VAR_INST
  _sResult,
  _sCtrl            : STRING(30);

  _stMsg            : ST_Message;
END_VAR

  _stMsg.eType               := E_MessageType.eMessageInfo;
  _stMsg.eDevice             := E_Device.NciChannelCtrl + TO_UINT(ChnId);
  _stMsg.eSubdevice          := e_Subdevice.NciControl;
  _stMsg.iErrorNumber        := 0;

  _sCtrl                     := concat('E_NCI_CTRL', '.');
  _sCtrl                     := concat(_sCtrl, TO_STRING(_eCtrlOld));

  _sResult                   := concat(': E_PROGRESS', '.');
  _sResult                   := concat(_sResult, TO_STRING(_eResult));

  _stMsg.sText               := concat(_sCtrl, ' ');
  _stMsg.sText               := concat(_sCtrl, _sResult);

  IF (_MessageLevel < E_MessageType.eMessageError)
  THEN
    f_MessageSet(_stMsg);
  ELSE
    IF (_stMsg.eType = E_MessageType.eMessageError)
    THEN
      f_MessageSet(_stMsg);
    END_IF
  END_IF
END_METHOD

PROPERTY M_FunctionScope : pointer to st_nci_m_func
SET
_MFuncScope := M_FunctionScope;
END_SET
END_PROPERTY

METHOD Template : E_PROGRESS
VAR_INPUT
  Execute           : BOOL;
END_VAR
VAR_INST
  _eState           : E_PROGRESS;
  _rValue           : LREAL;
  _udiErr           : UDINT;
  _stMsg            : ST_Message;


END_VAR
IF NOT Check() THEN _eState := E_PROGRESS.ERROR; END_IF
IF NOT Execute THEN _eState := E_PROGRESS.INIT; END_IF

CASE _eState
OF
  E_PROGRESS.INIT:
    IF Execute 
    THEN
      memset(ADR(_stMsg),0,SIZEOF(_stMsg));
      _udiErr                       := 0;
      _rValue                       := 0;
      _eState                       := E_PROGRESS.BUSY;
    END_IF
END_CASE
CASE _eState
OF
  E_PROGRESS.BUSY:
    _eState                         := E_PROGRESS.STARTUP;
END_CASE
CASE _eState
OF
  E_PROGRESS.STARTUP:
    _eState                       := E_PROGRESS.PREPARE;
END_CASE
CASE _eState
OF
  E_PROGRESS.PREPARE:
    _eState                         := E_PROGRESS.READY;
END_CASE
CASE _eState
OF
  E_PROGRESS.READY:
    _eState                         := E_PROGRESS.WAITING;
END_CASE
CASE _eState
OF
  E_PROGRESS.WAITING:
    _eState                         := E_PROGRESS.WORKING;
END_CASE
CASE _eState
OF
  E_PROGRESS.WORKING:
    _eState                         := E_PROGRESS.DONE;
END_CASE

Template_1 := _eState;
END_METHOD

END_FUNCTION_BLOCK

// ---- NCI/FB_NciChannel.TcPOU
FUNCTION_BLOCK FB_NciChannel IMPLEMENTS I_NciChannel
VAR
  ChannelDevice         : e_Device := e_Device.NciChannel;

// 2nd result of Check()
  _eCheck               : E_CHECK_STATE;

  _MessageLevel         : E_MessageType;

//NCI-Channel reference
  _NciChannelRef        : POINTER TO ST_NciChannel_Ref;

//Configured Group Axes
  _stCfgAxes            : POINTER TO ST_3D_Group;

//NCI-Group
  _fbBuildGroup         : Tc2_NCI.CfgBuildExt3DGroup;
  _fbClearGroup         : Tc2_NCI.CfgReconfigGroup;

  _fOverride            : LREAL := 100;

  _mdx,
  _adx                  : UINT;
  
//NCI-Program
{IF defined (WIN)}
  _sProg                : STRING(255) := 'C:\TwinCAT\Mc\Nci\Test_GST.nc';
{ELSE}
  _sProg                : STRING(255) := '/usr/local/etc/TwinCAT/Mc/Nci/Test_GST.nc';
{END_IF}

  _fbLoadProg           : Tc2_NCI.ItpLoadProgEx;

//Interpreter
  _fbReset              : Tc2_NCI.ItpResetEx2;
  _fbStartStop          : Tc2_NCI.ItpStartStopEx;
  _fbEStop              : Tc2_NCI.ItpEStopEx;
  _fbStepOnAfterEStop   : Tc2_NCI.ItpStepOnAfterEStopEx;

  _fbItpConfirmHsk      : Tc2_NCI.ItpConfirmHsk;
  _fbItpReadRParams     : Tc2_NCI.ItpReadRParamsEx;
  _fbItpWriteRParams    : Tc2_NCI.ItpWriteRParamsEx;
  _fbItpDelDtg          : Tc2_NCI.ItpDelDtgEx;

//ADS-Communication
  _fbReadLine           : Tc2_System.ADSREADEX;

// R Parameter
  // R[] Params used in G-Code
  // R[0..899]    local namespace of Channel
  // R[900..999]  global namespace of NC
  _pParameterRead       : POINTER TO ST_R_Parameter;
  _pParameterWrite      : POINTER TO ST_R_Parameter;
END_VAR

METHOD BuilDGroup : E_PROGRESS
VAR_INPUT
  Execute           : BOOL;
END_VAR
VAR_INST
  _eState           : E_PROGRESS;
  _rValue           : LREAL;
  _udiErr           : UDINT;
  _stMsg            : ST_Message;
END_VAR
IF NOT Check() THEN BuilDGroup := E_PROGRESS.ERROR; RETURN; END_IF
IF NOT Execute THEN _eState := E_PROGRESS.INIT; END_IF

CASE _eState
OF
  E_PROGRESS.INIT:
    IF Execute 
    THEN
      _fbBuildGroup( 
                bExecute            := FALSE, 
                nGroupId            := ItpGetGroupId(sNciToPlc:=_NciChannelRef^.NcToPlc) , 
                nXAxisId            := _stCfgAxes^.nXAxisId,
                nYAxisId            := _stCfgAxes^.nYAxisId, 
                nZAxisId            := _stCfgAxes^.nZAxisId, 
                nQ1AxisId           := _stCfgAxes^.nQ1AxisId,
                nQ2AxisId           := _stCfgAxes^.nQ2AxisId, 
                nQ3AxisId           := _stCfgAxes^.nQ3AxisId, 
                nQ4AxisId           := _stCfgAxes^.nQ4AxisId, 
                nQ5AxisId           := _stCfgAxes^.nQ5AxisId);

      memset(ADR(_stMsg),0,SIZEOF(_stMsg));
      _udiErr                       := 0;
      _rValue                       := 0;
      _eState                       := E_PROGRESS.BUSY;
    END_IF
END_CASE
CASE _eState
OF
  E_PROGRESS.BUSY:
    _eState                         := E_PROGRESS.STARTUP;
    _fbBuildGroup( 
                bExecute            := TRUE, 
                nGroupId            := ItpGetGroupId(sNciToPlc:=_NciChannelRef^.NcToPlc),
                  nErrId            => _udiErr);

    IF _fbBuildGroup.bErr 
    THEN
      _eState                       := E_PROGRESS.ERROR;

      _stMsg.eType                  := E_MessageType.eMessageError;
      _stMsg.eDevice                := ChannelDevice;
      _stMsg.eSubdevice             := e_Subdevice.fbBuildGroup;
      _stMsg.iErrorNumber           := _fbBuildGroup.nErrId;
      _stMsg.sText                  := concat('BuildGroup Error: ', TO_STRING(_fbBuildGroup.nErrId));
      f_MessageSet(_stMsg);

    ELSE
      IF _fbBuildGroup.bBusy
      THEN
        _eState                     := E_PROGRESS.STARTUP;

        _stMsg.eType                := E_MessageType.eMessageInfo;
        _stMsg.eDevice              := ChannelDevice;
        _stMsg.eSubdevice           := e_Subdevice.fbBuildGroup;
        _stMsg.iErrorNumber         := _fbBuildGroup.nGroupId;
        _stMsg.sText                := concat('BuildGroup Busy: ', TO_STRING(_fbBuildGroup.nGroupId));

        IF (_MessageLevel < E_MessageType.eMessageError)
        THEN
          f_MessageSet(_stMsg);
        END_IF
      END_IF
    END_IF
END_CASE
CASE _eState
OF
  E_PROGRESS.STARTUP:
    _fbBuildGroup( 
                bExecute            := TRUE, 
                nGroupId            := ItpGetGroupId(sNciToPlc:=_NciChannelRef^.NcToPlc),
                  nErrId            => _udiErr);

    IF _fbBuildGroup.bErr 
    THEN
      _eState                       := E_PROGRESS.ERROR;

      _stMsg.eType                  := E_MessageType.eMessageError;
      _stMsg.eDevice                := ChannelDevice;
      _stMsg.eSubdevice             := e_Subdevice.fbBuildGroup;
      _stMsg.iErrorNumber           := _fbBuildGroup.nErrId;
      _stMsg.sText                  := concat('BuildGroup Error: ', TO_STRING(_fbBuildGroup.nErrId));
      f_MessageSet(_stMsg);

    ELSE
      IF NOT _fbBuildGroup.bBusy
      THEN
        _eState                     := E_PROGRESS.DONE;

        _stMsg.eType                := E_MessageType.eMessageInfo;
        _stMsg.eDevice              := ChannelDevice;
        _stMsg.eSubdevice           := e_Subdevice.fbBuildGroup;
        _stMsg.iErrorNumber         := _fbBuildGroup.nGroupId;
        _stMsg.sText                := concat('BuildGroup Done: ', TO_STRING(_fbBuildGroup.nGroupId));

        IF (_MessageLevel < E_MessageType.eMessageError)
        THEN
          f_MessageSet(_stMsg);
        END_IF
      END_IF
    END_IF
END_CASE
CASE _eState
OF
  E_PROGRESS.ERROR,
  E_PROGRESS.DONE:
    _fbBuildGroup( 
                bExecute            := FALSE, 
                nGroupId            := ItpGetGroupId(sNciToPlc:=_NciChannelRef^.NcToPlc));
END_CASE


BuilDGroup                          := _eState;
END_METHOD

(*
===============================================================
NCI-Group configured axes structure
===============================================================
*)
PROPERTY CfgAxes : POINTER TO ST_3D_Group
SET
_stCfgAxes := CfgAxes;  //Configured Group Axes
END_SET
END_PROPERTY

PROPERTY ChannelRef : POINTER TO ST_NciChannel_Ref
SET
_NciChannelRef := ChannelRef;
END_SET
END_PROPERTY

METHOD Check : BOOL
VAR
  _idx      : uint;
END_VAR
IF NOT NCI_ACTIVE
THEN
  _eCheck                         := E_CHECK_STATE.NCI_NOT_ACTIVATED;
  RETURN;
END_IF

IF NOT (_NciChannelRef <> 0)
THEN
  _eCheck                         := E_CHECK_STATE.NCI_CHANNEL_REF_POINTER_INVALID;
  RETURN;
END_IF

IF NOT (_NciChannelRef^.NcToPlc.ChnId <> 0)
THEN
  _eCheck                         := E_CHECK_STATE.NCI_CHANNEL_REF_POINTER_INVALID;
  RETURN;
END_IF

IF (_stCfgAxes <> 0)
THEN
  _eCheck                         := E_CHECK_STATE.NCI_AXIS_CONFIG_POINTER_INVALID;
  RETURN;
END_IF

IF NOT (_pParameterRead <> 0)
THEN
  _eCheck                         := E_CHECK_STATE.NCI_R_PARAMETER_READ_POINTER_INVALID;
  RETURN;
END_IF

IF NOT (_pParameterWrite <> 0)
THEN
  _eCheck                         := E_CHECK_STATE.NCI_R_PARAMETER_WRITE_POINTER_INVALID;
  RETURN;
END_IF

_eCheck                           := E_CHECK_STATE.CHECK_DONE;
Check                             := TRUE;
END_METHOD

METHOD ClearGroup : E_PROGRESS
VAR_INPUT
  Execute           : BOOL;
END_VAR
VAR_INST
  _eState           : E_PROGRESS;
  _rValue           : LREAL;
  _udiErr           : UDINT;
  _stMsg            : ST_Message;
END_VAR
IF NOT Check() THEN ClearGroup := E_PROGRESS.ERROR; RETURN; END_IF
IF NOT Execute THEN _eState := E_PROGRESS.INIT; END_IF

CASE _eState
OF
  E_PROGRESS.INIT:
    IF Execute 
    THEN
      _fbClearGroup( 
                  bExecute          := FALSE, 
                  nGroupId          := ItpGetGroupId(sNciToPlc:= _NciChannelRef^.NcToPlc));

      memset(ADR(_stMsg),0,SIZEOF(_stMsg));
      _udiErr                       := 0;
      _rValue                       := 0;
      _eState                       := E_PROGRESS.BUSY;
    END_IF
END_CASE
CASE _eState
OF
  E_PROGRESS.BUSY:
    _eState                         := E_PROGRESS.STARTUP;
    _fbClearGroup( 
                  bExecute          := TRUE, 
                  nGroupId          := ItpGetGroupId(sNciToPlc:= _NciChannelRef^.NcToPlc),
                  nErrId            => _udiErr);

    IF _fbClearGroup.bErr 
    THEN
      _eState                       := E_PROGRESS.ERROR;

      _stMsg.eType                  := E_MessageType.eMessageError;
      _stMsg.eDevice                := ChannelDevice;
      _stMsg.eSubdevice             := e_Subdevice.fbClearGroup;
      _stMsg.iErrorNumber           := _fbClearGroup.nErrId;
      _stMsg.sText                  := concat('ClearGroup Error: ', TO_STRING(_fbClearGroup.nErrId));
      f_MessageSet(_stMsg);

    ELSE
      IF _fbClearGroup.bBusy
      THEN
        _eState                     := E_PROGRESS.STARTUP;
        _stMsg.eType                := E_MessageType.eMessageInfo;
        _stMsg.eDevice              := ChannelDevice;
        _stMsg.eSubdevice           := e_Subdevice.fbClearGroup;
        _stMsg.iErrorNumber         := _fbClearGroup.nErrId;
        _stMsg.sText                := concat('ClearGroup Busy: ', TO_STRING(_fbClearGroup.nErrId));

        IF (_MessageLevel < E_MessageType.eMessageError)
        THEN
          f_MessageSet(_stMsg);
        END_IF
      END_IF
    END_IF
END_CASE
CASE _eState
OF
  E_PROGRESS.STARTUP:
    _fbClearGroup( 
                  bExecute          := TRUE, 
                  nGroupId          := ItpGetGroupId(sNciToPlc:= _NciChannelRef^.NcToPlc),
                  nErrId            => _udiErr);

    IF _fbClearGroup.bErr 
    THEN
      _eState                       := E_PROGRESS.ERROR;

      _stMsg.eType                  := E_MessageType.eMessageError;
      _stMsg.eDevice                := ChannelDevice;
      _stMsg.eSubdevice             := e_Subdevice.fbClearGroup;
      _stMsg.iErrorNumber           := _fbClearGroup.nErrId;
      _stMsg.sText                  := concat('ClearGroup Error: ', TO_STRING(_fbClearGroup.nErrId));
      f_MessageSet(_stMsg);

    ELSE
      IF NOT _fbClearGroup.bBusy
      THEN
        _eState                     := E_PROGRESS.PREPARE;

        _stMsg.eType                := E_MessageType.eMessageInfo;
        _stMsg.eDevice              := ChannelDevice;
        _stMsg.eSubdevice           := e_Subdevice.fbClearGroup;
        _stMsg.iErrorNumber         := _fbClearGroup.nErrId;
        _stMsg.sText                := concat('ClearGroup Done: ', TO_STRING(_fbClearGroup.nErrId));

        IF (_MessageLevel < E_MessageType.eMessageError)
        THEN
          f_MessageSet(_stMsg);
        END_IF
      END_IF
    END_IF
END_CASE
CASE _eState
OF
  E_PROGRESS.PREPARE:
    _eState                         := E_PROGRESS.READY;
END_CASE
CASE _eState
OF
  E_PROGRESS.READY:
    _eState                         := E_PROGRESS.WAITING;
END_CASE
CASE _eState
OF
  E_PROGRESS.WAITING:
    _eState                         := E_PROGRESS.WORKING;
END_CASE
CASE _eState
OF
  E_PROGRESS.WORKING:
    _eState                         := E_PROGRESS.DONE;
END_CASE
CASE _eState
OF
  E_PROGRESS.ERROR,
  E_PROGRESS.DONE:
    _fbClearGroup( 
                  bExecute          := FALSE, 
                  nGroupId          := ItpGetGroupId(sNciToPlc:= _NciChannelRef^.NcToPlc));
END_CASE


ClearGroup                          := _eState;
END_METHOD

METHOD ConfirmHSK : E_PROGRESS
VAR_INPUT
  Execute           : BOOL;
END_VAR
VAR_INST
  _eState           : E_PROGRESS;
  _rValue           : LREAL;
  _udiErr           : UDINT;
  _stMsg            : ST_Message;
END_VAR
IF NOT Check() THEN ConfirmHSK := E_PROGRESS.ERROR; RETURN; END_IF
IF NOT Execute THEN _eState := E_PROGRESS.INIT; END_IF

CASE _eState
OF
  E_PROGRESS.INIT:
    _NciChannelRef^.PlcToNc.MFuncGranted   := 0;

    IF Execute 
    THEN
      memset(ADR(_stMsg),0,SIZEOF(_stMsg));
      _udiErr                                 := 0;
      _rValue                                 := 0;
      _eState                                 := E_PROGRESS.BUSY;
    END_IF
END_CASE
CASE _eState
OF
  E_PROGRESS.BUSY:
    IF (_NciChannelRef^.PlcToNc.ChnAxesOvr > 0) AND NOT
       (_NciChannelRef^.NcToPlc.ChnState.8)
    THEN
      IF (_NciChannelRef^.NcToPlc.HskMFuncReq = 1)
      THEN
        _eState                               := E_PROGRESS.STARTUP;

        _stMsg.eType                          := E_MessageType.eMessageInfo;
        _stMsg.eDevice                        := ChannelDevice;
        _stMsg.eSubdevice                     := e_Subdevice.fbConfirmHskItp;
        _stMsg.iErrorNumber                   := _NciChannelRef^.NcToPlc.HskMFuncNo;
        _stMsg.sText                          := concat('M Func check: ', 
                                                 TO_STRING(_NciChannelRef^.NcToPlc.HskMFuncNo));
        IF (_MessageLevel < E_MessageType.eMessageError)
        THEN
          f_MessageSet(_stMsg);
        END_IF
      END_IF
    END_IF
END_CASE
CASE _eState
OF
  E_PROGRESS.STARTUP:
    _NciChannelRef^.PlcToNc.MFuncGranted   := 1;

    IF (_NciChannelRef^.NcToPlc.HskMFuncReq = 0)
    THEN
      _eState                                 := E_PROGRESS.PREPARE;
      _NciChannelRef^.PlcToNc.MFuncGranted := 0;

      _stMsg.eType                            := E_MessageType.eMessageInfo;
      _stMsg.eDevice                          := ChannelDevice;
      _stMsg.eSubdevice                       := e_Subdevice.fbConfirmHskItp;
      _stMsg.iErrorNumber                     := _NciChannelRef^.NcToPlc.HskMFuncNo;
      _stMsg.sText                            := concat('M Func gone: ', 
                                               TO_STRING(_NciChannelRef^.NcToPlc.HskMFuncNo));
      IF (_MessageLevel < E_MessageType.eMessageError)
      THEN
        f_MessageSet(_stMsg);
      END_IF
    END_IF
END_CASE
CASE _eState
OF
  E_PROGRESS.PREPARE:
    _eState                         := E_PROGRESS.READY;
END_CASE
CASE _eState
OF
  E_PROGRESS.READY:
    _eState                         := E_PROGRESS.WAITING;
END_CASE
CASE _eState
OF
  E_PROGRESS.WAITING:
    _eState                         := E_PROGRESS.WORKING;
END_CASE
CASE _eState
OF
  E_PROGRESS.WORKING:
    _eState                         := E_PROGRESS.DONE;
END_CASE


ConfirmHSK                          := _eState;
END_METHOD

METHOD DeleteDistanceToGo : E_PROGRESS
VAR_INPUT
  Execute           : BOOL;
END_VAR
VAR_INST
  _eState           : E_PROGRESS;
  _rValue           : LREAL;
  _udiErr           : UDINT;
  _stMsg            : ST_Message;
END_VAR
IF NOT Check() THEN DeleteDistanceToGo := E_PROGRESS.ERROR; RETURN; END_IF
IF NOT Execute THEN _eState := E_PROGRESS.INIT; END_IF

CASE _eState
OF
  E_PROGRESS.INIT:
    _fbItpDelDtg(
                sNciToPlc   := _NciChannelRef^.NcToPlc, 
                bExecute    := FALSE);

    IF Execute 
    THEN
      memset(ADR(_stMsg),0,SIZEOF(_stMsg));
      _udiErr                                 := 0;
      _rValue                                 := 0;
      _eState                                 := E_PROGRESS.BUSY;
    END_IF
END_CASE
CASE _eState
OF
  E_PROGRESS.BUSY:
    _fbItpDelDtg(
                sNciToPlc   := _NciChannelRef^.NcToPlc, 
                bExecute    := TRUE,
                nErrId      => _udiErr);

    IF _fbItpDelDtg.bErr 
    THEN
      _eState                       := E_PROGRESS.ERROR;

      _stMsg.eType                  := E_MessageType.eMessageError;
      _stMsg.eDevice                := ChannelDevice;
      _stMsg.eSubdevice             := e_Subdevice.fbDelDtgItp;
      _stMsg.iErrorNumber           := _fbItpDelDtg.nErrId;
      _stMsg.sText                  := concat('Delete DistanceToGo Error: ', TO_STRING(_fbItpDelDtg.nErrId));
      f_MessageSet(_stMsg);

    ELSE
      IF _fbItpDelDtg.bBusy
      THEN
        _eState                     := E_PROGRESS.STARTUP;

        _stMsg.eType                := E_MessageType.eMessageInfo;
        _stMsg.eDevice              := ChannelDevice;
        _stMsg.eSubdevice           := e_Subdevice.fbDelDtgItp;
        _stMsg.iErrorNumber         := _fbItpDelDtg.nErrId;
        _stMsg.sText                := concat('Delete DistanceToGo Busy: ', TO_STRING(_fbItpDelDtg.nErrId));

        IF (_MessageLevel < E_MessageType.eMessageError)
        THEN
          f_MessageSet(_stMsg);
        END_IF
      END_IF
    END_IF
END_CASE
CASE _eState
OF
  E_PROGRESS.STARTUP:
    _fbItpDelDtg(
                sNciToPlc   := _NciChannelRef^.NcToPlc, 
                bExecute    := TRUE,
                nErrId      => _udiErr);

    IF _fbItpDelDtg.bErr 
    THEN
      _eState                       := E_PROGRESS.ERROR;

      _stMsg.eType                  := E_MessageType.eMessageError;
      _stMsg.eDevice                := ChannelDevice;
      _stMsg.eSubdevice             := e_Subdevice.fbDelDtgItp;
      _stMsg.iErrorNumber           := _fbItpDelDtg.nErrId;
      _stMsg.sText                  := concat('Delete DistanceToGo Error: ', TO_STRING(_fbItpDelDtg.nErrId));
      f_MessageSet(_stMsg);

    ELSE
      IF NOT _fbItpDelDtg.bBusy
      THEN
        _eState                     := E_PROGRESS.PREPARE;

        _stMsg.eType                := E_MessageType.eMessageInfo;
        _stMsg.eDevice              := ChannelDevice;
        _stMsg.eSubdevice           := e_Subdevice.fbDelDtgItp;
        _stMsg.iErrorNumber         := _fbItpDelDtg.nErrId;
        _stMsg.sText                := concat('Delete DistanceToGo Done: ', TO_STRING(_fbItpDelDtg.nErrId));
        f_MessageSet(_stMsg);
      END_IF
    END_IF
END_CASE
CASE _eState
OF
  E_PROGRESS.PREPARE:
    _eState                         := E_PROGRESS.READY;
END_CASE
CASE _eState
OF
  E_PROGRESS.READY:
    _eState                         := E_PROGRESS.WAITING;
END_CASE
CASE _eState
OF
  E_PROGRESS.WAITING:
    _eState                         := E_PROGRESS.WORKING;
END_CASE
CASE _eState
OF
  E_PROGRESS.WORKING:
    _eState                         := E_PROGRESS.DONE;
END_CASE
CASE _eState
OF
  E_PROGRESS.ERROR,
  E_PROGRESS.DONE:
    _fbItpDelDtg(
                sNciToPlc   := _NciChannelRef^.NcToPlc, 
                bExecute    := FALSE);
END_CASE


DeleteDistanceToGo                  := _eState;
END_METHOD

(*
===============================================================
Error-Flag
===============================================================
*)
PROPERTY Error : BOOL
GET
// get error from channel state
Error:= Error_Get();
END_GET
END_PROPERTY

METHOD Error_Get : BOOL
VAR_INST
  _stMsg            : ST_Message;
END_VAR
IF NOT Check() THEN RETURN; END_IF

//NciChannel
IF _NciChannelRef^.NcToPlc.ErrorCode <> 0 
THEN
  _stMsg.eType         := E_MessageType.eMessageError;
  _stMsg.eDevice       := ChannelDevice;
  _stMsg.eSubdevice    := e_Subdevice.Get_Error;
  _stMsg.iErrorNumber  := _NciChannelRef^.NcToPlc.ErrorCode;
  _stMsg.sText         := concat('NCI-Error: ', TO_STRING(_NciChannelRef^.NcToPlc.ErrorCode));
  f_MessageSet(_stMsg);

  Error_Get           := TRUE;
END_IF
END_METHOD

METHOD EStop : E_PROGRESS
VAR_INPUT
  Execute           : BOOL;
END_VAR
VAR_INST
  _eState           : E_PROGRESS;
  _rValue           : LREAL;
  _udiErr           : UDINT;
  _stMsg            : ST_Message;
END_VAR
IF NOT Check() THEN EStop := E_PROGRESS.ERROR; RETURN; END_IF
IF NOT Execute THEN _eState := E_PROGRESS.INIT; END_IF

CASE _eState
OF
  E_PROGRESS.INIT:
    _fbEStop(
            sNciToPlc               := _NciChannelRef^.NcToPlc, 
            bExecute                := FALSE);

    IF Execute 
    THEN
      memset(ADR(_stMsg),0,SIZEOF(_stMsg));
      _udiErr                       := 0;
      _rValue                       := 0;
      _eState                       := E_PROGRESS.BUSY;
    END_IF
END_CASE
CASE _eState
OF
  E_PROGRESS.BUSY:
    _fbEStop(
            sNciToPlc               := _NciChannelRef^.NcToPlc, 
            bExecute                := TRUE,
                nErrId              => _udiErr);

    IF _fbEStop.bErr 
    THEN
      _eState                       := E_PROGRESS.ERROR;

      _stMsg.eType                  := E_MessageType.eMessageError;
      _stMsg.eDevice                := ChannelDevice;
      _stMsg.eSubdevice             := e_Subdevice.fbEStopItp;
      _stMsg.iErrorNumber           := _fbEStop.nErrId;
      _stMsg.sText                  := concat('E-StopItp Error: ', TO_STRING(_fbEStop.nErrId));
      f_MessageSet(_stMsg);

    ELSE
      IF _fbEStop.bBusy
      THEN
        _eState                     := E_PROGRESS.STARTUP;

        _stMsg.eType                := E_MessageType.eMessageInfo;
        _stMsg.eDevice              := ChannelDevice;
        _stMsg.eSubdevice           := e_Subdevice.fbEStopItp;
        _stMsg.iErrorNumber         := _fbEStop.nErrId;
        _stMsg.sText                := concat('E-StopItp Busy: ', TO_STRING(_fbEStop.nErrId));

        IF (_MessageLevel < E_MessageType.eMessageError)
        THEN
          f_MessageSet(_stMsg);
        END_IF
      END_IF
    END_IF
END_CASE
CASE _eState
OF
  E_PROGRESS.STARTUP:
    _fbEStop(
            sNciToPlc               := _NciChannelRef^.NcToPlc, 
            bExecute                := TRUE,
                nErrId              => _udiErr);

    IF _fbEStop.bErr 
    THEN
      _eState                       := E_PROGRESS.ERROR;

      _stMsg.eType                  := E_MessageType.eMessageError;
      _stMsg.eDevice                := ChannelDevice;
      _stMsg.eSubdevice             := e_Subdevice.fbEStopItp;
      _stMsg.iErrorNumber           := _fbEStop.nErrId;
      _stMsg.sText                  := concat('E-StopItp Error: ', TO_STRING(_fbEStop.nErrId));
      f_MessageSet(_stMsg);

    ELSE
      IF NOT _fbEStop.bBusy
      THEN
        _eState                     := E_PROGRESS.PREPARE;

        _stMsg.eType                := E_MessageType.eMessageInfo;
        _stMsg.eDevice              := ChannelDevice;
        _stMsg.eSubdevice           := e_Subdevice.fbEStopItp;
        _stMsg.iErrorNumber         := _fbEStop.nErrId;
        _stMsg.sText                := concat('E-StopItp Done: ', TO_STRING(_fbEStop.nErrId));
        f_MessageSet(_stMsg);
      END_IF
    END_IF
END_CASE
CASE _eState
OF
  E_PROGRESS.PREPARE:
    _eState                         := E_PROGRESS.READY;
END_CASE
CASE _eState
OF
  E_PROGRESS.READY:
    _eState                         := E_PROGRESS.WAITING;
END_CASE
CASE _eState
OF
  E_PROGRESS.WAITING:
    _eState                         := E_PROGRESS.WORKING;
END_CASE
CASE _eState
OF
  E_PROGRESS.WORKING:
    _eState                         := E_PROGRESS.DONE;
END_CASE
CASE _eState
OF
  E_PROGRESS.ERROR,
  E_PROGRESS.DONE:
    _fbEStop(
            sNciToPlc               := _NciChannelRef^.NcToPlc, 
            bExecute                := FALSE);
END_CASE


EStop                               := _eState;
END_METHOD

METHOD GetChannelOverride : real
VAR_INPUT
END_VAR
IF NOT Check() THEN RETURN; END_IF
GetChannelOverride := TO_REAL(_NciChannelRef^.PlcToNc.ChnAxesOvr)/10_000.0;
END_METHOD

METHOD GetItpState : uint
VAR_INPUT
END_VAR
IF NOT Check() THEN RETURN; END_IF
GetItpState := _NciChannelRef^.NcToPlc.ItpState;
END_METHOD

METHOD GetLoadedProg : string
VAR_INPUT
END_VAR
GetLoadedProg := _fbLoadProg.sPrg;
END_METHOD

(*
===============================================================
Handshake: Announce and acknowledge M-Functions
===============================================================
*)
PROPERTY HSK : BOOL
GET

HSK :=  TO_BOOL(_NciChannelRef^.NcToPlc.HskMFuncReq);
END_GET
END_PROPERTY

PROPERTY ItpAxes : ST_3D_Group
GET
VAR
  stItpAxes     : ST_3D_Group;
END_VAR

stItpAxes.nXAxisId  := _NciChannelRef^.NcToPlc.AcsAxisIDs[0];
stItpAxes.nYAxisId  := _NciChannelRef^.NcToPlc.AcsAxisIDs[1];
stItpAxes.nZAxisId  := _NciChannelRef^.NcToPlc.AcsAxisIDs[2];
stItpAxes.nQ1AxisId := _NciChannelRef^.NcToPlc.AcsAxisIDs[3];
stItpAxes.nQ2AxisId := _NciChannelRef^.NcToPlc.AcsAxisIDs[4];
stItpAxes.nQ3AxisId := _NciChannelRef^.NcToPlc.AcsAxisIDs[5];
stItpAxes.nQ4AxisId := _NciChannelRef^.NcToPlc.AcsAxisIDs[6];
stItpAxes.nQ5AxisId := _NciChannelRef^.NcToPlc.AcsAxisIDs[7];

ItpAxes := stItpAxes;
END_GET
END_PROPERTY

METHOD ItpReset   : E_PROGRESS
VAR_INPUT
  Execute           : BOOL;
END_VAR
VAR_INST
  _eState           : E_PROGRESS;
  _rValue           : LREAL;
  _udiErr           : UDINT;
  _stMsg            : ST_Message;
END_VAR
IF NOT Check() THEN ItpReset := E_PROGRESS.ERROR; RETURN; END_IF
IF NOT Execute THEN _eState := E_PROGRESS.INIT; END_IF

CASE _eState
OF
  E_PROGRESS.INIT:
    _fbReset(
            bExecute                := FALSE, 
            tTimeOut                := T#1S, 
            sNciToPlc               := _NciChannelRef^.NcToPlc);

    IF Execute 
    THEN
      memset(ADR(_stMsg),0,SIZEOF(_stMsg));
      _udiErr                       := 0;
      _rValue                       := 0;
      _eState                       := E_PROGRESS.BUSY;
    END_IF
END_CASE
CASE _eState
OF
  E_PROGRESS.BUSY:
    _fbReset(
            bExecute                := TRUE, 
            tTimeOut                := T#1S, 
            sNciToPlc               := _NciChannelRef^.NcToPlc,
               nErrId               => _udiErr);

    IF _fbReset.bErr 
    THEN
      _eState                       := E_PROGRESS.ERROR;

      _stMsg.eType                  := E_MessageType.eMessageError;
      _stMsg.eDevice                := ChannelDevice;
      _stMsg.eSubdevice             := e_Subdevice.fbResetItp;
      _stMsg.iErrorNumber           := _fbReset.nErrId;
      _stMsg.sText                  := concat('ResetItp Error: ', TO_STRING(_fbReset.nErrId));
      f_MessageSet(_stMsg);

    ELSE
//      IF _fbReset.bBusy
//      THEN
        _eState                     := E_PROGRESS.STARTUP;

        _stMsg.eType                := E_MessageType.eMessageInfo;
        _stMsg.eDevice              := ChannelDevice;
        _stMsg.eSubdevice           := e_Subdevice.fbResetItp;
        _stMsg.iErrorNumber         := _fbReset.nErrId;
        _stMsg.sText                := concat('ResetItp Busy: ', TO_STRING(_fbReset.nErrId));

        IF (_MessageLevel < E_MessageType.eMessageError)
        THEN
          f_MessageSet(_stMsg);
        END_IF
      END_IF
//    END_IF
END_CASE
CASE _eState
OF
  E_PROGRESS.STARTUP:
    _fbReset(
            bExecute                := TRUE, 
            tTimeOut                := T#1S, 
            sNciToPlc               := _NciChannelRef^.NcToPlc,
               nErrId               => _udiErr);

    IF _fbReset.bErr 
    THEN
      _eState                       := E_PROGRESS.ERROR;

      _stMsg.eType                  := E_MessageType.eMessageError;
      _stMsg.eDevice                := ChannelDevice;
      _stMsg.eSubdevice             := e_Subdevice.fbResetItp;
      _stMsg.iErrorNumber           := _fbReset.nErrId;
      _stMsg.sText                  := concat('ResetItp Error: ', TO_STRING(_fbReset.nErrId));
      f_MessageSet(_stMsg);

    ELSE
      IF NOT _fbReset.bBusy
      THEN
        _eState                     := E_PROGRESS.PREPARE;

        _stMsg.eType                := E_MessageType.eMessageInfo;
        _stMsg.eDevice              := ChannelDevice;
        _stMsg.eSubdevice           := e_Subdevice.fbResetItp;
        _stMsg.iErrorNumber         := _fbReset.nErrId;
        _stMsg.sText                := concat('ResetItp Done: ', TO_STRING(_fbReset.nErrId));
        f_MessageSet(_stMsg);
      END_IF
    END_IF
END_CASE
CASE _eState
OF
  E_PROGRESS.PREPARE:
    _eState                         := E_PROGRESS.READY;
END_CASE
CASE _eState
OF
  E_PROGRESS.READY:
    _eState                         := E_PROGRESS.WAITING;
END_CASE
CASE _eState
OF
  E_PROGRESS.WAITING:
    _eState                         := E_PROGRESS.WORKING;
END_CASE
CASE _eState
OF
  E_PROGRESS.WORKING:
    _eState                         := E_PROGRESS.DONE;
END_CASE
CASE _eState
OF
  E_PROGRESS.ERROR,
  E_PROGRESS.DONE:
    _fbReset(
            bExecute                := FALSE, 
            tTimeOut                := T#1S, 
            sNciToPlc               := _NciChannelRef^.NcToPlc);
END_CASE


ItpReset                            := _eState;
END_METHOD

METHOD LoadProg   : E_PROGRESS
VAR_INPUT
  Execute           : BOOL;
END_VAR
VAR_INST
  _eState           : E_PROGRESS;
  _rValue           : LREAL;
  _udiErr           : UDINT;
  _stMsg            : ST_Message;
END_VAR
IF NOT Check() THEN LoadProg := E_PROGRESS.ERROR; RETURN; END_IF
IF NOT Execute THEN _eState := E_PROGRESS.INIT; END_IF

CASE _eState
OF
  E_PROGRESS.INIT:
    _fbLoadProg(
               sNciToPlc            := _NciChannelRef^.NcToPlc, 
               bExecute             := FALSE, 
               sPrg                 := _sProg, 
               nLength              := TO_UDINT(LEN(_sProg)));

    IF Execute 
    THEN
      memset(ADR(_stMsg),0,SIZEOF(_stMsg));
      _udiErr                       := 0;
      _rValue                       := 0;
      _eState                       := E_PROGRESS.BUSY;
    END_IF
END_CASE
CASE _eState
OF
  E_PROGRESS.BUSY:
    _fbLoadProg(
               sNciToPlc            := _NciChannelRef^.NcToPlc, 
               bExecute             := TRUE, 
               sPrg                 := _sProg, 
               nLength              := TO_UDINT(LEN(_sProg)),
               nErrId               => _udiErr);

    IF _fbLoadProg.bErr 
    THEN
      _eState                       := E_PROGRESS.ERROR;

      _stMsg.eType                  := E_MessageType.eMessageError;
      _stMsg.eDevice                := ChannelDevice;
      _stMsg.eSubdevice             := e_Subdevice.fbLoadProg;
      _stMsg.iErrorNumber           := _fbLoadProg.nErrId;
      _stMsg.sText                  := concat('LoadProg Error: ', TO_STRING(_fbLoadProg.nErrId));
      f_MessageSet(_stMsg);

    ELSE
      IF _fbLoadProg.bBusy
      THEN
        _eState                     := E_PROGRESS.STARTUP;

        _stMsg.eType                := E_MessageType.eMessageInfo;
        _stMsg.eDevice              := ChannelDevice;
        _stMsg.eSubdevice           := e_Subdevice.fbLoadProg;
        _stMsg.iErrorNumber         := _fbLoadProg.nErrId;
        _stMsg.sText                := concat('LoadProg Busy: ', TO_STRING(_fbLoadProg.nErrId));

        IF (_MessageLevel < E_MessageType.eMessageError)
        THEN
          f_MessageSet(_stMsg);
        END_IF
      END_IF
    END_IF
END_CASE
CASE _eState
OF
  E_PROGRESS.STARTUP:
    _fbLoadProg(
               sNciToPlc            := _NciChannelRef^.NcToPlc, 
               bExecute             := TRUE, 
               sPrg                 := _sProg, 
               nLength              := TO_UDINT(LEN(_sProg)),
               nErrId               => _udiErr);

    IF _fbLoadProg.bErr 
    THEN
      _eState                       := E_PROGRESS.ERROR;

      _stMsg.eType                  := E_MessageType.eMessageError;
      _stMsg.eDevice                := ChannelDevice;
      _stMsg.eSubdevice             := e_Subdevice.fbLoadProg;
      _stMsg.iErrorNumber           := _fbLoadProg.nErrId;
      _stMsg.sText                  := concat('Load Prog Error: ', TO_STRING(_fbLoadProg.nErrId));
      f_MessageSet(_stMsg);

    ELSE
      IF NOT _fbLoadProg.bBusy
      THEN
        _eState                     := E_PROGRESS.PREPARE;

        _stMsg.eType                := E_MessageType.eMessageInfo;
        _stMsg.eDevice              := ChannelDevice;
        _stMsg.eSubdevice           := e_Subdevice.fbLoadProg;
        _stMsg.iErrorNumber         := _fbLoadProg.nErrId;
        _stMsg.sText                := concat('Load Prog Done: ', TO_STRING(_fbLoadProg.nErrId));

        IF (_MessageLevel < E_MessageType.eMessageError)
        THEN
          f_MessageSet(_stMsg);
        END_IF
      END_IF
    END_IF
END_CASE
CASE _eState
OF
  E_PROGRESS.PREPARE:
    IF (_NciChannelRef^.NcToPlc.ItpState = Tc2_NCI.NCI_INTERPRETER_READY)
    THEN
      _eState                       := E_PROGRESS.READY;

    ELSIF (_NciChannelRef^.NcToPlc.ItpState = Tc2_NCI.NCI_INTERPRETER_ABORTED)
    THEN
      _eState                       := E_PROGRESS.ERROR;

      _stMsg.eType                  := E_MessageType.eMessageError;
      _stMsg.eDevice                := ChannelDevice;
      _stMsg.eSubdevice             := e_Subdevice.fbLoadProg;
      _stMsg.iErrorNumber           := _NciChannelRef^.NcToPlc.ErrorCode;
      _stMsg.sText                  := concat('Chn State: ', TO_STRING(_NciChannelRef^.NcToPlc.ChnState));
      f_MessageSet(_stMsg);

    END_IF
END_CASE
CASE _eState
OF
  E_PROGRESS.READY:
    _eState                         := E_PROGRESS.WAITING;
END_CASE
CASE _eState
OF
  E_PROGRESS.WAITING:
    _eState                         := E_PROGRESS.WORKING;
END_CASE
CASE _eState
OF
  E_PROGRESS.WORKING:
    _eState                         := E_PROGRESS.DONE;
END_CASE
CASE _eState
OF
  E_PROGRESS.ERROR,
  E_PROGRESS.DONE:
    _fbLoadProg(
               sNciToPlc            := _NciChannelRef^.NcToPlc, 
               bExecute             := FALSE, 
               sPrg                 := _sProg, 
               nLength              := TO_UDINT(LEN(_sProg)));
END_CASE

LoadProg                            := _eState;
END_METHOD

PROPERTY M_FuncReq : word
GET
M_FuncReq := _NciChannelRef^.NcToPlc.HskMFuncReq;
END_GET
END_PROPERTY

PROPERTY MessageLevel : E_MessageType
SET
_MessageLevel := MessageLevel;
END_SET
END_PROPERTY

(*
===============================================================
M-Function
===============================================================
*)
PROPERTY MFunc : INT
GET

MFunc := TO_INT(_NciChannelRef^.NcToPlc.HskMFuncNo);
END_GET
END_PROPERTY

PROPERTY Override : LREAL
GET
Override := Tc2_NCI.ItpGetOverridePercent(_NciChannelRef^.PlcToNc);
END_GET
SET
Tc2_NCI.ItpSetOverridePercent(Override, _NciChannelRef^.PlcToNc);
END_SET
END_PROPERTY

(*
===============================================================
actual path velo [Units/s]
===============================================================
*)
PROPERTY PathVelo : LREAL
GET

PathVelo := _NciChannelRef^.NcToPlc.PathVelo;
END_GET
END_PROPERTY

(*
===============================================================
G-Code Program Name (sFilePath)
===============================================================
*)
PROPERTY Prog : STRING(255)
GET
Prog:=_sProg;
END_GET
SET
_sProg:=Prog;
END_SET
END_PROPERTY

PROPERTY R_ParameterRead : Pointer to ST_R_Parameter;
SET
_pParameterRead := R_ParameterRead;
END_SET
END_PROPERTY

PROPERTY R_ParameterWrite : pointer to ST_R_Parameter;
SET
_pParameterWrite := R_ParameterWrite;
END_SET
END_PROPERTY

METHOD ReadLine   : E_PROGRESS
VAR_INPUT
  Execute           : BOOL;
END_VAR
//Read G-Code actual Line
VAR_OUTPUT
  ActProgLine       : STRING(100);
END_VAR
VAR_INST
  _ReadString       : STRING(100);
  _nBlockNo         : UDINT;

  _eState           : E_PROGRESS;
  _rValue           : LREAL;
  _udiErr           : UDINT;
  _stMsg            : ST_Message;
END_VAR
IF NOT Check() THEN ReadLine := E_PROGRESS.ERROR; RETURN; END_IF
IF NOT Execute THEN _eState := E_PROGRESS.INIT; END_IF

CASE _eState
OF
  E_PROGRESS.INIT:
    _fbReadLine(
               PORT                 := 500, 
               IDXGRP               := 16#2300 + _NciChannelRef^.NcToPlc.ChnId, // + ChannelID
               IDXOFFS              := 16#2000_0001,
               LEN                  := SIZEOF(_ReadString),
               DESTADDR             := ADR(_ReadString), 
               READ                 := FALSE);

    IF Execute 
    THEN
      memset(ADR(_ReadString),0,SIZEOF(_ReadString));
      memset(ADR(_stMsg),     0,SIZEOF(_stMsg));
      _udiErr                       := 0;
      _rValue                       := 0;
      _eState                       := E_PROGRESS.BUSY;
    END_IF
END_CASE
CASE _eState
OF
  E_PROGRESS.BUSY:
    _fbReadLine(
               PORT                 := 500, 
               IDXGRP               := 16#2300 + _NciChannelRef^.NcToPlc.ChnId, // + ChannelID
               IDXOFFS              := 16#2000_0001,
               LEN                  := SIZEOF(_ReadString),
               DESTADDR             := ADR(_ReadString), 
               READ                 := TRUE);

    IF _fbReadLine.ERR 
    THEN
      _eState                       := E_PROGRESS.ERROR;

      _stMsg.eType                  := E_MessageType.eMessageError;
      _stMsg.eDevice                := ChannelDevice;
      _stMsg.eSubdevice             := e_Subdevice.fbReadLine;
      _stMsg.iErrorNumber           := _fbReadLine.ERRID;
      _stMsg.sText                  := concat('ReadLine Error: ', TO_STRING(_fbReadLine.ERRID));
      f_MessageSet(_stMsg);

    ELSE
      IF _fbReadLine.BUSY
      THEN
        _eState                     := E_PROGRESS.STARTUP;

        _stMsg.eType                := E_MessageType.eMessageInfo;
        _stMsg.eDevice              := ChannelDevice;
        _stMsg.eSubdevice           := e_Subdevice.fbReadLine;
        _stMsg.iErrorNumber         := _fbReadLine.ERRID;
        _stMsg.sText                := concat('ReadLine Busy: ', TO_STRING(_fbReadLine.ERRID));

        IF (_MessageLevel < E_MessageType.eMessageError)
        THEN
          f_MessageSet(_stMsg);
        END_IF
      END_IF
    END_IF
END_CASE
CASE _eState
OF
  E_PROGRESS.STARTUP:
    _fbReadLine(
               PORT                 := 500, 
               IDXGRP               := 16#2300 + _NciChannelRef^.NcToPlc.ChnId, // + ChannelID
               IDXOFFS              := 16#2000_0001,
               LEN                  := SIZEOF(_ReadString),
               DESTADDR             := ADR(_ReadString), 
               READ                 := TRUE);

    IF _fbReadLine.ERR 
    THEN
      _eState                       := E_PROGRESS.ERROR;

      _stMsg.eType                  := E_MessageType.eMessageError;
      _stMsg.eDevice                := ChannelDevice;
      _stMsg.eSubdevice             := e_Subdevice.fbReadLine;
      _stMsg.iErrorNumber           := _fbReadLine.ERRID;
      _stMsg.sText                  := concat('ReadLine Error: ', TO_STRING(_fbReadLine.ERRID));
      f_MessageSet(_stMsg);

    ELSE
      IF NOT _fbReadLine.BUSY
      THEN
        ActProgLine                 := _ReadString;

        _eState                     := E_PROGRESS.PREPARE;

        _stMsg.eType                := E_MessageType.eMessageInfo;
        _stMsg.eDevice              := ChannelDevice;
        _stMsg.eSubdevice           := e_Subdevice.fbReadLine;
        _stMsg.iErrorNumber         := _fbReadLine.ERRID;
        _stMsg.sText                := concat('ReadLine Done: ', TO_STRING(_fbReadLine.ERRID));

        IF (_MessageLevel < E_MessageType.eMessageError)
        THEN
          f_MessageSet(_stMsg);
        END_IF
      END_IF
    END_IF
END_CASE
CASE _eState
OF
  E_PROGRESS.PREPARE:
    _eState                         := E_PROGRESS.READY;
END_CASE
CASE _eState
OF
  E_PROGRESS.READY:
    _eState                         := E_PROGRESS.WAITING;
END_CASE
CASE _eState
OF
  E_PROGRESS.WAITING:
    _eState                         := E_PROGRESS.WORKING;
END_CASE
CASE _eState
OF
  E_PROGRESS.WORKING:
    _eState                         := E_PROGRESS.DONE;
END_CASE
CASE _eState
OF
  E_PROGRESS.ERROR,
  E_PROGRESS.DONE:
    _fbReadLine(
               PORT                 := 500, 
               IDXGRP               := 16#2300 + _NciChannelRef^.NcToPlc.ChnId, // + ChannelID
               IDXOFFS              := 16#2000_0001,
               LEN                  := SIZEOF(_ReadString),
               DESTADDR             := ADR(_ReadString), 
               READ                 := FALSE);
END_CASE


ReadLine                            := _eState;
END_METHOD

METHOD ReadRParams : E_PROGRESS
VAR_INPUT
  Execute  : BOOL;
END_VAR
VAR_INST
  _eState           : E_PROGRESS;
  _udiErr           : UDINT;
  _stMsg            : ST_Message;

  // local copy of last successful read
  _nIndex           : DINT;
  _nCount           : DINT;
  _rValue           : ARRAY[0..MAX_R_PARA] OF LREAL;
END_VAR
IF NOT Check() THEN ReadRParams := E_PROGRESS.ERROR; RETURN; END_IF
IF NOT Execute THEN _eState := E_PROGRESS.INIT; END_IF

CASE _eState
OF
  E_PROGRESS.INIT:
    IF Execute 
    THEN
      memset(ADR(_stMsg),  0,SIZEOF(_stMsg));
      memset(ADR(_rValue), 0,SIZEOF(_rValue));

      _udiErr := _nIndex := _nCount := 0;
      _eState                       := E_PROGRESS.BUSY;

      _fbItpReadRParams(
                  sNciToPlc         := _NciChannelRef^.NcToPlc, 
                  bExecute          := FALSE, 
                  pAddr             := ADR(_rValue), 
                  nIndex            := _pParameterRead^._nStart, 
                  nCount            := _pParameterRead^._nCount);
    END_IF
END_CASE
CASE _eState
OF
  E_PROGRESS.BUSY:
    _fbItpReadRParams(
                  sNciToPlc         := _NciChannelRef^.NcToPlc, 
                  bExecute          := TRUE, 
                  pAddr             := ADR(_rValue), 
                  nIndex            := _pParameterRead^._nStart, 
                  nCount            := _pParameterRead^._nCount,
                  nErrId            => _udiErr);

    IF _fbItpReadRParams.bErr 
    THEN
      _eState                       := E_PROGRESS.ERROR;

      _stMsg.eType                  := E_MessageType.eMessageError;
      _stMsg.eDevice                := ChannelDevice;
      _stMsg.eSubdevice             := e_Subdevice.fbItpReadRParams;
      _stMsg.iErrorNumber           := _fbItpReadRParams.nErrId;
      _stMsg.sText                  := concat('Read R Parameter Error: ', TO_STRING(_fbItpReadRParams.nErrId));
      f_MessageSet(_stMsg);

    ELSE
      IF _fbItpReadRParams.bBusy
      THEN
        _eState                     := E_PROGRESS.PREPARE;

        _stMsg.eType                := E_MessageType.eMessageInfo;
        _stMsg.eDevice              := ChannelDevice;
        _stMsg.eSubdevice           := e_Subdevice.fbItpReadRParams;
        _stMsg.iErrorNumber         := _fbItpReadRParams.nErrId;
        _stMsg.sText                := concat('Read R Parameter Busy: ', TO_STRING(_fbItpReadRParams.nErrId));
        IF (_MessageLevel < E_MessageType.eMessageError)
        THEN
          f_MessageSet(_stMsg);
        END_IF
      END_IF
    END_IF
END_CASE
CASE _eState
OF
  E_PROGRESS.STARTUP:
    _fbItpReadRParams(
                  sNciToPlc         := _NciChannelRef^.NcToPlc, 
                  bExecute          := TRUE, 
                  pAddr             := ADR(_rValue), 
                  nIndex            := _pParameterRead^._nStart, 
                  nCount            := _pParameterRead^._nCount,
                  nErrId            => _udiErr);

    IF _fbItpReadRParams.bErr 
    THEN
      _eState                       := E_PROGRESS.ERROR;

      _stMsg.eType                  := E_MessageType.eMessageError;
      _stMsg.eDevice                := ChannelDevice;
      _stMsg.eSubdevice             := e_Subdevice.fbItpReadRParams;
      _stMsg.iErrorNumber           := _fbItpReadRParams.nErrId;
      _stMsg.sText                  := concat('Read R Parameter Error: ', TO_STRING(_fbItpReadRParams.nErrId));
      f_MessageSet(_stMsg);

    ELSE
      IF NOT _fbItpReadRParams.bBusy
      THEN
        _eState                     := E_PROGRESS.PREPARE;

        _stMsg.eType                := E_MessageType.eMessageInfo;
        _stMsg.eDevice              := ChannelDevice;
        _stMsg.eSubdevice           := e_Subdevice.fbItpReadRParams;
        _stMsg.iErrorNumber         := _fbItpReadRParams.nErrId;
        _stMsg.sText                := concat('Read R Parameter Done: ', TO_STRING(_fbItpReadRParams.nErrId));
        IF (_MessageLevel < E_MessageType.eMessageError)
        THEN
          f_MessageSet(_stMsg);
        END_IF
      END_IF
    END_IF
END_CASE
CASE _eState
OF
  E_PROGRESS.PREPARE:
    _nIndex                         := _pParameterRead^._nStart;
    _nCount                         := _pParameterRead^._nCount;
    _pParameterRead^._rValue        := _rValue;

    _eState                         := E_PROGRESS.DONE;
END_CASE
CASE _eState
OF
  E_PROGRESS.ERROR,
  E_PROGRESS.DONE:
    _fbItpReadRParams(
                  sNciToPlc         := _NciChannelRef^.NcToPlc, 
                  bExecute          := FALSE, 
                  pAddr             := ADR(_pParameterRead^._rValue), 
                  nIndex            := _pParameterRead^._nStart, 
                  nCount            := _pParameterRead^._nCount);
END_CASE


ReadRParams                         := _eState;
END_METHOD

METHOD StartStop : E_PROGRESS
VAR_INPUT
  Execute           : BOOL;
  Start             : BOOL;
  Stop              : BOOL;
END_VAR
VAR_INST
  _eState           : E_PROGRESS;
  _rValue           : LREAL;
  _udiErr           : UDINT;
  _stMsg            : ST_Message;
END_VAR
IF NOT Check() THEN StartStop := E_PROGRESS.ERROR; RETURN; END_IF
IF NOT Execute THEN _eState := E_PROGRESS.INIT; END_IF

CASE _eState
OF
  E_PROGRESS.INIT:
    _fbStartStop(
                bStart              := FALSE, 
                bStop               := FALSE, 
                sNciToPlc           := _NciChannelRef^.NcToPlc);

    IF Execute 
    THEN
      memset(ADR(_stMsg),0,SIZEOF(_stMsg));
      _udiErr                       := 0;
      _rValue                       := 0;
      _eState                       := E_PROGRESS.BUSY;
    END_IF
END_CASE
CASE _eState
OF
  E_PROGRESS.BUSY:
    _fbStartStop(
                bStart              := Start, 
                bStop               := Stop, 
                sNciToPlc           := _NciChannelRef^.NcToPlc,
                nErrId              => _udiErr);

    IF _fbStartStop.bErr 
    THEN
      _eState                       := E_PROGRESS.ERROR;

      _stMsg.eType                  := E_MessageType.eMessageError;
      _stMsg.eDevice                := ChannelDevice;
      _stMsg.eSubdevice             := e_Subdevice.fbStartStopItp;
      _stMsg.iErrorNumber           := _fbStartStop.nErrId;
      _stMsg.sText                  := concat('StartStop Itp Error: ', TO_STRING(_fbStartStop.nErrId));
      f_MessageSet(_stMsg);

    ELSE
      IF _fbStartStop.bBusy
      THEN
        _eState                     := E_PROGRESS.STARTUP;

